// TIA Portal project "SCI_prueba_485" (V17)

(* hardware
DEVICE "ET 200SP station_1"  ET 200SP-Station
   slot 0: "Rack_0"  Rack  6ES5 710-8MAx1
   slot 1: "PLC_1"  CPU 1510SP-1 PN  6ES7 510-1DJ01-0AB0  V2.9
      slot 32768: "Interfaz PROFINET_1"  X1
   slot 2: "CM PtP_1"  CM PtP  6ES7 137-6AA01-0BA0  V2.0
      slot 1: "CM PtP_1"  CM PtP Sub
   slot 3: "Módulo servidor_1"  Server module  6ES7 193-6PA00-0AA0  V1.1
      slot 1: "Módulo servidor_1"  Server module
   slot 127: "BA 2xRJ45"  BA 2xRJ45  6ES7 193-6AR00-0AA0  V0.0
      slot 32769: "Port_1"  6ES7 193-6AR00-0AA0
      slot 32770: "Port_2"  6ES7 193-6AR00-0AA0
*)

// ===== PLC "PLC_1"  CPU 1510SP-1 PN =====

VAR_GLOBAL   // PLC tag table "Tabla de variables estándar"
   "System_Byte" AT %MB1 : Byte;
   "FirstScan" AT %M1.0 : Bool;
   "DiagStatusUpdate" AT %M1.1 : Bool;
   "AlwaysTRUE" AT %M1.2 : Bool;
   "AlwaysFALSE" AT %M1.3 : Bool;
   "Clock_Byte" AT %MB0 : Byte;
   "Clock_10Hz" AT %M0.0 : Bool;
   "Clock_5Hz" AT %M0.1 : Bool;
   "Clock_2.5Hz" AT %M0.2 : Bool;
   "Clock_2Hz" AT %M0.3 : Bool;
   "Clock_1.25Hz" AT %M0.4 : Bool;
   "Clock_1Hz" AT %M0.5 : Bool;
   "Clock_0.625Hz" AT %M0.6 : Bool;
   "Clock_0.5Hz" AT %M0.7 : Bool;
   "Tag_1" AT %MD100 : DWord;
   "Tag_2" AT %M50.0 : Bool;
   "Tag_3" AT %M64.0 : Bool;
   "Tag_4" AT %M64.1 : Bool;
   "Tag_5" AT %M70.0 : Bool;
END_VAR

VAR_GLOBAL   // PLC tag table "IO"
   "ZS01" AT %I0.0 : Bool;   // Contacto Magnético P2-6
   "ZS02" AT %I0.1 : Bool;   // Contacto Magnético P2-5
   "ZS03" AT %I0.2 : Bool;   // Contacto Magnético P2-4
   "HS01" AT %I0.3 : Bool;   // Pulsador P2-6 A
   "HS02" AT %I0.4 : Bool;   // Pulsador P2-6 B
   "HS03" AT %I0.5 : Bool;   // Pulsador P2-5 A
   "HS04" AT %I0.6 : Bool;   // Pulsador P2-4 A
   "HSS01" AT %I0.7 : Bool;   // Puño de emergencia ducha
   "YY01" AT %I1.0 : Bool;   // Señal apertura del controlador puerta P2-5
   "YY02" AT %I1.1 : Bool;   // Señal apertura del controlador puerta P2-4
   "PSH01" AT %I1.2 : Bool;   // Presóstado burlete P2-6
   "E1.3" AT %I1.3 : Bool;   // Reserva
   "E1.4" AT %I1.4 : Bool;   // Reserva
   "E1.5" AT %I1.5 : Bool;   // Reserva
   "E1.6" AT %I1.6 : Bool;   // Reserva
   "E1.7" AT %I1.7 : Bool;   // Reserva
   "EV01" AT %A0.0 : Bool;   // Electroválvula ducha
   "KY01" AT %Q0.1 : Bool;   // PUERTA P2-6
   "KY02" AT %Q0.2 : Bool;   // PUERTA P2-5
   "KY03" AT %Q0.3 : Bool;   // PUERTA P2-4
   "HA01" AT %Q0.4 : Bool;   // P2-6 Buzzer - Hombre atrapado
   "HL01" AT %Q0.5 : Bool;   // P2-6 Lámpara - Falla
   "KY04" AT %Q0.6 : Bool;   // Reinicio fuente
   "Q0.7" AT %Q0.7 : Bool;   // Reserva
   "Q1.0" AT %Q1.0 : Bool;   // Reserva
   "Q1.1" AT %Q1.1 : Bool;   // Reserva
   "Q1.2" AT %Q1.2 : Bool;   // Reserva
   "Q1.3" AT %Q1.3 : Bool;   // Reserva
   "Q1.4" AT %Q1.4 : Bool;   // Reserva
   "Q1.5" AT %Q1.5 : Bool;   // Reserva
   "Q1.6" AT %Q1.6 : Bool;   // Reserva
   "Q1.7" AT %Q1.7 : Bool;   // Reserva
END_VAR

TYPE "FALLAS"
   STRUCT
      PE_FACT : Bool;   // Falla: Emergencia actuada
      Vestuario_FTMO : Bool;   // Falla: Persona en vestuario por demasiado tiempo
      Ducha_FTMO : Bool;   // Falla: Persona en ducha por demasiado tiempo
      "P2-6_FATR" : Bool;   // Falla: P2-6 Persona atrapada
      "P2-5_FATR" : Bool;   // Falla: P2-5 Persona atrapada
      "P2-4_FATR" : Bool;   // Falla: P2-4 Persona atrapada
      "P2-6_TMO_FABR" : Bool;   // Falla: Puerta P2-6 abierta
      "P2-5_TMO_FABR" : Bool;   // Falla: Puerta P2-5 abierta
      "P2-4_TMO_FABR" : Bool;   // Falla: Puerta P2-4 abierta
   END_STRUCT;
END_TYPE

DATA_BLOCK "DB1_AVISOS"   // DB1
TITLE = DB Avisos
{ S7_Optimized_Access := 'FALSE' }
AUTHOR : IGLP
VERSION : 0.1
   VAR
      PRE : "FALLAS";
      MEM : "FALLAS";
      REC : "FALLAS";
      CMD : "FALLAS";
      CMD_AUX : "FALLAS";
      CMD_FLA : "FALLAS";
   END_VAR
BEGIN
END_DATA_BLOCK

DATA_BLOCK "DB2_CODIGOS"   // DB2
TITLE = Códigos habilitados
{ S7_Optimized_Access := 'TRUE' }
AUTHOR : IGLP
VERSION : 0.1
   VAR
      PIN_Nuevo_TCL1 : Bool;
      PIN_Nuevo_TCL2 : Bool;
      PIN_TCL1_OK : Bool;
      PIN_TCL2_OK : Bool;
      PIN_TCL1_ERR : Bool;
      PIN_TCL2_ERR : Bool;
      PIN_Codigo_TCL1 : Int;
      PIN_Codigo_TCL2 : Int;
      PIN_Codigo_TCL1_OK : Int;
      PIN_Codigo_TCL2_OK : Int;
      Aux_inidice : Int;
      TCL1_TMR_BitVida : IEC_TIMER;
      TCL2_TMR_BitVida : IEC_TIMER;
      TCL_TMR_ESP : IEC_TIMER;
      TCL_PWR_OFF : IEC_TIMER;
   END_VAR
   VAR RETAIN
      PIN : Array[0..500] of Int;
   END_VAR
BEGIN
END_DATA_BLOCK

DATA_BLOCK "DB3_GRAL"   // DB3
TITLE = DB Comandos eléctricos
{ S7_Optimized_Access := 'TRUE' }
VERSION : 0.1
   VAR
      MODO : Int;   // Modo: 0 - Manual / 1 Automático
      REINICIO : Int;
      SILENCIAR : Int;
      CNT_Personas : Int;
      CNT_HS01 : Int;   // P2-6A: Cantidad de veces pulsado
      CNT_HS02 : Int;   // P2-6B: Cantidad de veces pulsado
      CNT_HS03 : Int;   // P2-5A: Cantidad de veces pulsado
      CNT_HS04 : Int;   // P2-4A: Cantidad de veces pulsado
      SFA : Bool;   // Sin fallas
      FNUE : Bool;   // Falla nueva
      FPRE : Bool;   // Falla presente
      "P2-x_ResFal" : Bool;   // Resumen de fallas de puerta
      fpHS01 : Bool;   // Flanco positivo - Pulsador P2-6 A
      fpHS02 : Bool;   // Flanco positivo - Pulsador P2-6 B
      fpHS03 : Bool;   // Flanco positivo - Pulsador P2-5 A
      fpHS04 : Bool;   // Flanco positivo - Pulsador P2-4 A
      xHS01 : Bool;
      xHS02 : Bool;
      xHS03 : Bool;
      xHS04 : Bool;
      xZS01 : Bool;
      xZS02 : Bool;
      xZS03 : Bool;
      xS161 : Bool;
      xS261 : Bool;
      TMR_TMO_Vestuario : IEC_TIMER;
      TMR_TMO_Ducha : IEC_TIMER;
      "TMR_P2-6_CRR" : IEC_TIMER;
      "TMR_P2-5_CRR" : IEC_TIMER;
      "TMR_P2-4_CRR" : IEC_TIMER;
      TMR_HS01_SCADA : IEC_TIMER;
      TMR_HS02_SCADA : IEC_TIMER;
      TMR_HS03_SCADA : IEC_TIMER;
      TMR_HS04_SCADA : IEC_TIMER;
      TMR_ZS01 : IEC_TIMER;
      TMR_ZS02 : IEC_TIMER;
      TMR_ZS03 : IEC_TIMER;
      TMR_PSH01 : IEC_TIMER;
      ZS01_TMP : Bool;   // Contacto Magnético P2-6 - Temporizado
      ZS02_TMP : Bool;   // Contacto Magnético P2-5 - Temporizado
      ZS03_TMP : Bool;   // Contacto Magnético P2-4 - Temporizado
      PSH01_TMP : Bool;   // Presóstado burlete P2-6 - Temporizado
      "P2-6" : Struct   // Puerta Pasillo <-> Vestuario P2-6
         TMR_Sol_Man : IEC_TIMER;
         Sol_Man : Bool;   // Solicitud manual de apertura
         HW : Bool;   // Hardware Interlock
         CMD : Bool;   // Comando de apertura
      END_STRUCT;
      "P2-5" : Struct   // Puerta Vestuario <-> Ducha P2-5
         TMR_Sol_Man : IEC_TIMER;
         Sol_Man : Bool;   // Solicitud manual de apertura
         HW : Bool;   // Hardware Interlock
         CMD : Bool;   // Comando de apertura
      END_STRUCT;
      "P2-4" : Struct   // Puerta Ducha <-> Bioterio P2-4
         TMR_Sol_Man : IEC_TIMER;
         Sol_Man : Bool;   // Solicitud manual de apertura
         HW : Bool;   // Hardware Interlock
         CMD : Bool;   // Comando de apertura
      END_STRUCT;
      Ducha : Struct   // Ducha - Electroválvula
         TMR_Sol_Man : IEC_TIMER;
         Sol_Man : Bool;   // Solicitud manual de apertura
         HW : Bool;   // Hardware Interlock
         CMD : Bool;
      END_STRUCT;
   END_VAR
BEGIN
END_DATA_BLOCK

DATA_BLOCK "DB10_Parámetros"   // DB10
TITLE = DB Parametros del sistema
{ S7_Optimized_Access := 'TRUE' }
AUTHOR : IGLP
VERSION : 0.1
   VAR RETAIN
      SP_N_APA : Int := 10;   // Consigna de veces antes de aviso persona atrapada
      SP_Tmp_Ducha_1 : DInt;   // Consigna de tiempo de ducha activa [ms]
      SP_Tmp_Ducha_2 : DInt := 30000;   // Consigna de tiempo de ducha activa [ms]
      SP_Tmp_Ducha_Pre : DInt;   // Consigna de tiempo de precalentar ducha [ms]
      SP_TMO_Ducha : DInt;   // Consigna de tiempo en ducha [ms]
      SP_TMO_Vestuario : DInt;   // Consigna de tiempo en vestuario [ms]
      SP_TMO_PTA_ABR : DInt;   // Consigna de tiempo alarma puerta abierta [ms]
   END_VAR
BEGIN
END_DATA_BLOCK

DATA_BLOCK "DB20_Modbus_Config"   // DB20
{ S7_Optimized_Access := 'TRUE' }
VERSION : 0.1
   VAR
      TC_NDR : Bool := FALSE;
      TC_DR : Bool := FALSE;
      TC_Error : Bool := FALSE;
      TC_Status : Word := 16#7000;
      SCADA_NDR : Bool := FALSE;
      SCADA_DR : Bool := FALSE;
      SCADA_Error : Bool := TRUE;
      SCADA_Status : Word := 16#8389;
      DATA : Array[0..1] of Int;
      SCADA_CONN : TCON_IP_v4;
   END_VAR
BEGIN
   SCADA_CONN.InterfaceId := 64;
   SCADA_CONN.ID := 16#001E;
   SCADA_CONN.ConnectionType := 16#0B;
   SCADA_CONN.LocalPort := 502;
   SCADA_CONN.RemotePort := 0;
   SCADA_CONN.ActiveEstablished := FALSE;
   SCADA_CONN.RemoteAddress.ADDR[1] := 0;
   SCADA_CONN.RemoteAddress.ADDR[2] := 0;
   SCADA_CONN.RemoteAddress.ADDR[3] := 0;
   SCADA_CONN.RemoteAddress.ADDR[4] := 0;
END_DATA_BLOCK

DATA_BLOCK "DB21_Modbus_Data_1"   // DB21
{ S7_Optimized_Access := 'FALSE' }
VERSION : 0.1
   VAR
      "NBS 3A" : Struct
         Modo : Int;   // Scada -> PLC: Modo (0-Manual / 1-Automático)
         Reinicio : Int;   // Scada -> PLC: Reset de secuencia
         Silenciar : Int;   // Scada -> PLC: Silenciar alarma
         SP_Tmp_Ducha : Int;   // Scada -> PLC: Consigna de tiempo de ducha activa [s]
         SP_Tmp_Ducha_Pre : Int;   // Scada -> PLC: Consigna de tiempo de precalentar ducha [s]
         SP_TMO_Ducha : Int;   // Scada -> PLC: Consigna de tiempo en ducha [s]
         SP_TMO_Vestuario : Int;   // Scada -> PLC: Consigna de tiempo en vestuario [s]
         SP_TMO_PTA_ABR : Int;   // Scada -> PLC: Consigna de tiempo alarma puerta abierta [s]
         CNT_Personas : Int;   // PLC -> Scada: Contador de personas dentro de bioterio
         "P2-6_Est" : Int;   // PLC -> Scada: P2-6 - Puerta Pasillo: Estado (0-Cerrada / 1-Abierta / 2-Falla reconocida / 3-Falla nueva)
         "P2-5_Est" : Int;   // PLC -> Scada: P2-5 - Puerta Ducha Ingreso: Estado (0-Cerrada / 1-Abierta / 2-Falla reconocida / 3-Falla nueva)
         "P2-4_Est" : Int;   // PLC -> Scada: P2-4 - Puerta Ducha Salida: Estado (0-Cerrada / 1-Abierta / 2-Falla reconocida / 3-Falla nueva)
         HSS01_Est : Int;   // PLC -> Scada: Pulsador de Emergencia en Ducha (0-Normal/ 1-Activada/ 2-Falla reconocida / 3-Falla nueva)
         HS01_Est : Int;   // PLC -> Scada: P2-6A: Pulsador Ingreso (0-Normal / 1-Presionado)
         HS02_Est : Int;   // PLC -> Scada: P2-6B: Pulsador Salida (0-Normal / 1-Presionado)
         HS03_Est : Int;   // PLC -> Scada: P2-5A: Pulsador Ducha Ingreso (0-Normal / 1-Presionado)
         HS04_Est : Int;   // PLC -> Scada: P2-4A: Pulsador Ducha Salida (0-Normal / 1-Presionado)
         EV01_Est : Int;   // PLC -> Scada: Ducha: Electroválvula (0-Normal/ 1-Activada/ 2-Falla reconocida / 3-Falla nueva)
         TCL01_PIN : Int;   // PLC -> Scada: P2-5: PIN ingresado en teclado
         TCL02_PIN : Int;   // PLC -> Scada: P2-6: PIN ingresado en teclado
         Ducha_PIN : Int;   // PLC -> Scada: Ducha: PIN de quien ingresó a ducha
         Vesuario_Est : Int;   // PLC -> Scada: Vestuario: Estado (0-Desocupado / 1-Ocupado / 2-Falla reconocida / 3-Falla nueva)
         Ducha_Est : Int;   // PLC -> Scada: Ducha: Estado (0-Desocupada / 1-Ocupada / 2-Falla reconocida / 3-Falla nueva)
         Alarma : Int;   // PLC -> Scada: Resumen de alarmas (0-Sin alarma / 1-Alarma presente)
      END_STRUCT;
   END_VAR
BEGIN
END_DATA_BLOCK

DATA_BLOCK "DB22_Modbus_Data_2"   // DB22
{ S7_Optimized_Access := 'FALSE' }
VERSION : 0.1
   VAR
      CODIGOS : Array[1..100] of Int;
   END_VAR
BEGIN
END_DATA_BLOCK

DATA_BLOCK "DB23_Modbus_Data_3"   // DB23
{ S7_Optimized_Access := 'FALSE' }
VERSION : 0.1
   VAR
      data : Array[0..10] of Int;
      TCL : Struct
         "TCL1 P2-5 PIN" : Int;
         "TCL1 P2-5 ALIVE" : Int;
         "TCL2 P2-4 PIN" : Int;
         "TCL2 P2-4 ALIVE" : Int;
      END_STRUCT;
   END_VAR
BEGIN
END_DATA_BLOCK

DATA_BLOCK "DB50_Secuencia"   // DB50
{ S7_Optimized_Access := 'TRUE' }
VERSION : 0.1
// stored: InstanceOfName Secuencia
"Secuencia"
BEGIN
END_DATA_BLOCK

DATA_BLOCK "DB51_Transiciones"   // DB51
TITLE = DB Transiciones y estados del secuencial
{ S7_Optimized_Access := 'TRUE' }
AUTHOR : IGLP
VERSION : 0.1
   VAR
      TMR_Puerta : IEC_TIMER;
      TMR_DUCHA_ESP_INI : IEC_TIMER;
      TMR_DUCHA_PRE : IEC_TIMER;
      TMR_DUCHA_1 : IEC_TIMER;
      TMR_DUCHA_2 : IEC_TIMER;
      TMR_DUCHA_3 : IEC_TIMER;
   END_VAR
   VAR RETAIN
      S : Struct
         "10" : Bool;   // Reposo
         "110" : Bool;   // Ingreso a bioterio: Solicitud ingreso Pasillo -> Vestuario
         "111" : Bool;   // Ingreso a bioterio: Puerta P2-6 abierta
         "120" : Bool;   // Ingreso a bioterio: Vestuario ocupado
         "121" : Bool;   // Ingreso a bioterio: Solicitud de precalentar ducha
         "130" : Bool;   // Ingreso a bioterio: Solicitud salir Vestuario -> Pasillo
         "131" : Bool;   // Ingreso a bioterio: Puerta P2-6 abierta
         "140" : Bool;   // Ingreso a bioterio: Solicitud ingreso Vestuario -> Ducha
         "141" : Bool;   // Ingreso a bioterio: Puerta P2-5 abierta
         "150" : Bool;   // Ingreso a bioterio: Ducha ocupada
         "160" : Bool;   // Ingreso a bioterio: Solicitud salir Ducha -> Bioterio
         "161" : Bool;   // Ingreso a bioterio: Puerta P2-4 abierta
         "170" : Bool;   // Ingreso a bioterio: Solicitud salir Ducha -> Vestuario
         "171" : Bool;   // Ingreso a bioterio: Puerta P2-5 abierta
         "210" : Bool;   // Egreso de bioterio: Solicitud ingreso Bioterio -> Ducha
         "211" : Bool;   // Egreso de bioterio: Puerta P2-4 abierta
         "220" : Bool;   // Egreso de bioterio: Ducha ocupada - Espera incial
         "221" : Bool;   // Egreso de bioterio: Ducha ocupada - Válvula abierta
         "222" : Bool;   // Egreso de bioterio: Ducha ocupada - Pausa ducha
         "223" : Bool;   // Egreso de bioterio: Ducha ocupada - Válvula abierta
         "224" : Bool;   // Egreso de bioterio: Ducha ocupada
         "230" : Bool;   // Egreso de bioterio: Solicitud salir Ducha -> Bioterio
         "231" : Bool;   // Egreso de bioterio: Puerta P2-4 abierta
         "240" : Bool;   // Egreso de bioterio: Solicitud salir Ducha -> Vestuario
         "241" : Bool;   // Egreso de bioterio: Puerta P2-5 abierta
         "250" : Bool;   // Egreso de bioterio: Vestuario ocupado
         "251" : Bool;   // Egreso de bioterio: Solicitud de precalentar ducha
         "260" : Bool;   // Egreso de bioterio: Solicitud salir Vestuario -> Pasillo
         "261" : Bool;   // Egreso de bioterio: Puerta P2-6 abierta
         "270" : Bool;   // Egreso de bioterio: Solicitud ingreso Vestuario -> Ducha
         "271" : Bool;   // Egreso de bioterio: Puerta P2-5 abierta
         "310" : Bool;   // Egreso de bioterio: Solicitud de precalentar ducha
      END_STRUCT;
   END_VAR
   VAR
      T : Struct
         T10_110 : Bool;
         T110_111 : Bool;
         T111_120 : Bool;
         T110_10 : Bool;
         T120_121 : Bool;
         T121_120 : Bool;
         T120_140 : Bool;
         T140_141 : Bool;
         T120_130 : Bool;
         T130_131 : Bool;
         T130_120 : Bool;
         T131_10 : Bool;
         T141_150 : Bool;
         T150_160 : Bool;
         T160_161 : Bool;
         T160_150 : Bool;
         T161_10 : Bool;
         T150_170 : Bool;
         T170_171 : Bool;
         T171_120 : Bool;
         T170_150 : Bool;
         T10_210 : Bool;
         T210_211 : Bool;
         T211_220 : Bool;
         T220_221 : Bool;
         T221_222 : Bool;
         T222_223 : Bool;
         T223_224 : Bool;
         T224_230 : Bool;
         T224_240 : Bool;
         T240_241 : Bool;
         T241_250 : Bool;
         T240_224 : Bool;
         T250_260 : Bool;
         T260_261 : Bool;
         T261_10 : Bool;
         T260_250 : Bool;
         T250_270 : Bool;
         T270_271 : Bool;
         T271_224 : Bool;
         T270_250 : Bool;
         T250_251 : Bool;
         T251_250 : Bool;
         T210_10 : Bool;
         T220_230 : Bool;
         T230_231 : Bool;
         T230_220 : Bool;
         T231_10 : Bool;
         T10_310 : Bool;
         T310_10 : Bool;
      END_STRUCT;
   END_VAR
BEGIN
END_DATA_BLOCK

FUNCTION_BLOCK "Secuencia"   // FB1, GRAPH_PLUS
{ S7_Optimized_Access := 'TRUE' }
VERSION : 0.1
   VAR_INPUT
      OFF_SQ : Bool := false;   // Desactivar cadena
      INIT_SQ : Bool := false;   // Poner cadena en estado inicial
      ACK_EF : Bool := false;   // Acusar todos los errores y fallos
      S_PREV : Bool := false;   // Mostrar la etapa anterior en el parámetro S_NO
      S_NEXT : Bool := false;   // Mostrar la etapa siguiente en el parámetro S_NO
      SW_AUTO : Bool := false;   // Modo automático
      SW_TAP : Bool := false;   // Semiautomático/continuar con transición
      SW_TOP : Bool := false;   // Semiautomático/transición ignorada
      SW_MAN : Bool := false;   // Modo manual
      S_SEL : Int := 0;   // Seleccionar la etapa que debe mostrarse en S_NO
      S_ON : Bool := false;   // Activar la etapa del parámetro S_NO
      S_OFF : Bool := false;   // Desactivar el incremento presente en el parámetro S_NO
      T_PUSH : Bool := false;   // Habilitar conmutación de transición en modo semiautomático
   END_VAR
   VAR_OUTPUT
      S_NO : Int := 0;   // Número de etapa
      S_MORE : Bool := false;   // Existen más etapas que pueden mostrarse en S_NO.
      S_ACTIVE : Bool := false;   // El incremento presente en el parámetro S_NO está activo
      ERR_FLT : Bool := false;   // Error de grupo interlock o supervisión
      AUTO_ON : Bool := false;   // Modo automático activado
      TAP_ON : Bool := false;   // Modo semiautomático/etapa con transición activada
      TOP_ON : Bool := false;   // Modo semiautomático/Ignorar transición activado
      MAN_ON : Bool := false;   // Modo manual activado
   END_VAR
   VAR
      HMI_INFO : Array[0..8] of UInt;
      IF_PAR : G7_IfParPlus_V6;
      RT_DATA : G7_RTDataPlus_V6;   // Área de datos interna
      T10_110 : G7_TransitionPlus_V6;   // Estructura de la transición
      T110_111 : G7_TransitionPlus_V6;   // Estructura de la transición
      T111_120 : G7_TransitionPlus_V6;   // Estructura de la transición
      T120_140 : G7_TransitionPlus_V6;   // Estructura de la transición
      T140_141 : G7_TransitionPlus_V6;   // Estructura de la transición
      T141_150 : G7_TransitionPlus_V6;   // Estructura de la transición
      T150_160 : G7_TransitionPlus_V6;   // Estructura de la transición
      T160_161 : G7_TransitionPlus_V6;   // Estructura de la transición
      T120_121 : G7_TransitionPlus_V6;   // Estructura de la transición
      T121_120 : G7_TransitionPlus_V6;   // Estructura de la transición
      T120_130 : G7_TransitionPlus_V6;   // Estructura de la transición
      T130_131 : G7_TransitionPlus_V6;   // Estructura de la transición
      T161_10 : G7_TransitionPlus_V6;   // Estructura de la transición
      T160_150 : G7_TransitionPlus_V6;   // Estructura de la transición
      T150_170 : G7_TransitionPlus_V6;   // Estructura de la transición
      T170_171 : G7_TransitionPlus_V6;   // Estructura de la transición
      T170_120 : G7_TransitionPlus_V6;   // Estructura de la transición
      T170_150 : G7_TransitionPlus_V6;   // Estructura de la transición
      T130_120 : G7_TransitionPlus_V6;   // Estructura de la transición
      T131_10 : G7_TransitionPlus_V6;   // Estructura de la transición
      T10_210 : G7_TransitionPlus_V6;   // Estructura de la transición
      T210_211 : G7_TransitionPlus_V6;   // Estructura de la transición
      T211_220 : G7_TransitionPlus_V6;   // Estructura de la transición
      T220_221 : G7_TransitionPlus_V6;   // Estructura de la transición
      T221_222 : G7_TransitionPlus_V6;   // Estructura de la transición
      T222_223 : G7_TransitionPlus_V6;   // Estructura de la transición
      T223_224 : G7_TransitionPlus_V6;   // Estructura de la transición
      T224_240 : G7_TransitionPlus_V6;   // Estructura de la transición
      S220_230 : G7_TransitionPlus_V6;   // Estructura de la transición
      S230_231 : G7_TransitionPlus_V6;   // Estructura de la transición
      T231_10 : G7_TransitionPlus_V6;   // Estructura de la transición
      S230_220 : G7_TransitionPlus_V6;   // Estructura de la transición
      T210_10 : G7_TransitionPlus_V6;   // Estructura de la transición
      T240_241 : G7_TransitionPlus_V6;   // Estructura de la transición
      T260_261 : G7_TransitionPlus_V6;   // Estructura de la transición
      T241_250 : G7_TransitionPlus_V6;   // Estructura de la transición
      T250_260 : G7_TransitionPlus_V6;   // Estructura de la transición
      T261_10 : G7_TransitionPlus_V6;   // Estructura de la transición
      T250_270 : G7_TransitionPlus_V6;   // Estructura de la transición
      T270_271 : G7_TransitionPlus_V6;   // Estructura de la transición
      T271_224 : G7_TransitionPlus_V6;   // Estructura de la transición
      T270_250 : G7_TransitionPlus_V6;   // Estructura de la transición
      T250_251 : G7_TransitionPlus_V6;   // Estructura de la transición
      T251_250 : G7_TransitionPlus_V6;   // Estructura de la transición
      T10_310 : G7_TransitionPlus_V6;   // Estructura de la transición
      T310_10 : G7_TransitionPlus_V6;   // Estructura de la transición
      T110_10 : G7_TransitionPlus_V6;   // Estructura de la transición
      T240_224 : G7_TransitionPlus_V6;   // Estructura de la transición
      T260_250 : G7_TransitionPlus_V6;   // Estructura de la transición
      T224_230 : G7_TransitionPlus_V6;   // Estructura de la transición
      Reposo : G7_StepPlus_V6;   // Estructura de la etapa
      S110 : G7_StepPlus_V6;   // Estructura de la etapa
      S111 : G7_StepPlus_V6;   // Estructura de la etapa
      S120 : G7_StepPlus_V6;   // Estructura de la etapa
      S121 : G7_StepPlus_V6;   // Estructura de la etapa
      S130 : G7_StepPlus_V6;   // Estructura de la etapa
      S131 : G7_StepPlus_V6;   // Estructura de la etapa
      S140 : G7_StepPlus_V6;   // Estructura de la etapa
      S141 : G7_StepPlus_V6;   // Estructura de la etapa
      S150 : G7_StepPlus_V6;   // Estructura de la etapa
      S160 : G7_StepPlus_V6;   // Estructura de la etapa
      S161 : G7_StepPlus_V6;   // Estructura de la etapa
      S170 : G7_StepPlus_V6;   // Estructura de la etapa
      S171 : G7_StepPlus_V6;   // Estructura de la etapa
      S210 : G7_StepPlus_V6;   // Estructura de la etapa
      S211 : G7_StepPlus_V6;   // Estructura de la etapa
      S220 : G7_StepPlus_V6;   // Estructura de la etapa
      S221 : G7_StepPlus_V6;   // Estructura de la etapa
      S222 : G7_StepPlus_V6;   // Estructura de la etapa
      S223 : G7_StepPlus_V6;   // Estructura de la etapa
      S224 : G7_StepPlus_V6;   // Estructura de la etapa
      S230 : G7_StepPlus_V6;   // Estructura de la etapa
      S231 : G7_StepPlus_V6;   // Estructura de la etapa
      S240 : G7_StepPlus_V6;   // Estructura de la etapa
      S241 : G7_StepPlus_V6;   // Estructura de la etapa
      S250 : G7_StepPlus_V6;   // Estructura de la etapa
      S251 : G7_StepPlus_V6;   // Estructura de la etapa
      S260 : G7_StepPlus_V6;   // Estructura de la etapa
      S261 : G7_StepPlus_V6;   // Estructura de la etapa
      S270 : G7_StepPlus_V6;   // Estructura de la etapa
      S271 : G7_StepPlus_V6;   // Estructura de la etapa
      S310 : G7_StepPlus_V6;   // Estructura de la etapa
      SINI : Array[0..1] of USInt;
      LSTT : Array[0..49] of USInt;
      ATAJ : Array[0..49] of USInt;
      ATAB : Array[0..49] of USInt;
      PSTT : Array[0..49] of USInt;
      NSTT : Array[0..49] of USInt;
      ASSJ : Array[0..31] of USInt;
      ASSB : Array[0..31] of USInt;
      PTTS : Array[0..31] of USInt;
      NTTS : Array[0..31] of USInt;
      SW_SQTS : Array[0..31] of USInt;
      SWITCH : Array[0..71] of USInt;
      TVX : Array[0..34] of USInt;
      TTX : Array[0..34] of USInt;
      TSX : Array[0..1] of USInt;
      S00X : Array[0..1] of USInt;
      SOFFX : Array[0..1] of USInt;
      SONX : Array[0..1] of USInt;
      SAX : Array[0..1] of USInt;
      SERRX : Array[0..32] of USInt;
      SMX : Array[0..32] of USInt;
      S0X : Array[0..32] of USInt;
      S1X : Array[0..32] of USInt;
      IL_ALARM_INST : Diag_Alarm;
      SUP_ALARM_INST : Diag_Alarm;
      STEP_TIME_ALARM_INST : Diag_Alarm;
      IEC_TIMER_INST : IEC_TIMER;
      TRANSACTION_FLAG : Bool := false;
   END_VAR
   // SINI[0] := 2;
   // LSTT[0] := 255;
   // LSTT[1] := 255;
   // LSTT[2] := 255;
   // LSTT[3] := 255;
   // LSTT[4] := 255;
   // LSTT[5] := 255;
   // LSTT[6] := 255;
   // LSTT[7] := 255;
   // LSTT[8] := 255;
   // LSTT[9] := 3;
   // LSTT[10] := 255;
   // LSTT[11] := 255;
   // LSTT[13] := 9;
   // LSTT[14] := 255;
   // LSTT[15] := 255;
   // LSTT[16] := 3;
   // LSTT[17] := 9;
   // LSTT[18] := 3;
   // LSTT[20] := 255;
   // LSTT[21] := 255;
   // LSTT[22] := 255;
   // LSTT[23] := 255;
   // LSTT[24] := 255;
   // LSTT[25] := 255;
   // LSTT[26] := 255;
   // LSTT[27] := 255;
   // LSTT[28] := 255;
   // LSTT[29] := 255;
   // LSTT[31] := 16;
   // LSTT[33] := 255;
   // LSTT[34] := 255;
   // LSTT[35] := 255;
   // LSTT[36] := 255;
   // LSTT[38] := 255;
   // LSTT[39] := 255;
   // LSTT[40] := 20;
   // LSTT[41] := 25;
   // LSTT[42] := 255;
   // LSTT[43] := 25;
   // LSTT[44] := 255;
   // ATAJ[1] := 1;
   // ATAJ[2] := 2;
   // ATAJ[3] := 3;
   // ATAJ[4] := 4;
   // ATAJ[5] := 5;
   // ATAJ[6] := 6;
   // ATAJ[7] := 7;
   // ATAJ[8] := 8;
   // ATAJ[9] := 9;
   // ATAJ[10] := 10;
   // ATAJ[11] := 11;
   // ATAJ[12] := 12;
   // ATAJ[13] := 13;
   // ATAJ[14] := 14;
   // ATAJ[15] := 15;
   // ATAJ[16] := 16;
   // ATAJ[17] := 17;
   // ATAJ[18] := 18;
   // ATAJ[19] := 19;
   // ATAJ[20] := 20;
   // ATAJ[21] := 21;
   // ATAJ[22] := 22;
   // ATAJ[23] := 23;
   // ATAJ[24] := 24;
   // ATAJ[25] := 25;
   // ATAJ[26] := 26;
   // ATAJ[27] := 27;
   // ATAJ[28] := 28;
   // ATAJ[29] := 29;
   // ATAJ[30] := 30;
   // ATAJ[31] := 31;
   // ATAJ[32] := 32;
   // ATAJ[33] := 33;
   // ATAJ[34] := 34;
   // ATAJ[35] := 35;
   // ATAJ[36] := 36;
   // ATAJ[37] := 37;
   // ATAJ[38] := 38;
   // ATAJ[39] := 39;
   // ATAJ[40] := 40;
   // ATAJ[41] := 41;
   // ATAJ[42] := 42;
   // ATAJ[43] := 43;
   // ATAJ[44] := 44;
   // ATAJ[45] := 45;
   // ATAB[0] := 20;
   // ATAB[1] := 46;
   // ATAB[2] := 2;
   // ATAB[3] := 8;
   // ATAB[4] := 4;
   // ATAB[5] := 5;
   // ATAB[6] := 14;
   // ATAB[7] := 13;
   // ATAB[8] := 10;
   // ATAB[9] := 9;
   // ATAB[10] := 3;
   // ATAB[11] := 18;
   // ATAB[12] := 12;
   // ATAB[13] := 7;
   // ATAB[14] := 6;
   // ATAB[15] := 17;
   // ATAB[16] := 16;
   // ATAB[17] := 15;
   // ATAB[18] := 11;
   // ATAB[19] := 19;
   // ATAB[20] := 44;
   // ATAB[21] := 32;
   // ATAB[22] := 22;
   // ATAB[23] := 28;
   // ATAB[24] := 24;
   // ATAB[25] := 25;
   // ATAB[26] := 26;
   // ATAB[27] := 49;
   // ATAB[28] := 23;
   // ATAB[29] := 31;
   // ATAB[30] := 30;
   // ATAB[31] := 29;
   // ATAB[32] := 21;
   // ATAB[33] := 47;
   // ATAB[34] := 48;
   // ATAB[35] := 35;
   // ATAB[36] := 38;
   // ATAB[37] := 37;
   // ATAB[38] := 42;
   // ATAB[39] := 41;
   // ATAB[40] := 40;
   // ATAB[41] := 39;
   // ATAB[42] := 36;
   // ATAB[43] := 43;
   // ATAB[45] := 45;
   // PSTT[1] := 1;
   // PSTT[2] := 2;
   // PSTT[3] := 3;
   // PSTT[4] := 7;
   // PSTT[5] := 8;
   // PSTT[6] := 9;
   // PSTT[7] := 10;
   // PSTT[8] := 3;
   // PSTT[9] := 4;
   // PSTT[10] := 3;
   // PSTT[11] := 5;
   // PSTT[12] := 11;
   // PSTT[13] := 10;
   // PSTT[14] := 9;
   // PSTT[15] := 12;
   // PSTT[16] := 13;
   // PSTT[17] := 12;
   // PSTT[18] := 5;
   // PSTT[19] := 6;
   // PSTT[21] := 14;
   // PSTT[22] := 15;
   // PSTT[23] := 16;
   // PSTT[24] := 17;
   // PSTT[25] := 18;
   // PSTT[26] := 19;
   // PSTT[27] := 20;
   // PSTT[28] := 16;
   // PSTT[29] := 21;
   // PSTT[30] := 22;
   // PSTT[31] := 21;
   // PSTT[32] := 14;
   // PSTT[33] := 23;
   // PSTT[34] := 27;
   // PSTT[35] := 24;
   // PSTT[36] := 25;
   // PSTT[37] := 28;
   // PSTT[38] := 25;
   // PSTT[39] := 29;
   // PSTT[40] := 30;
   // PSTT[41] := 29;
   // PSTT[42] := 25;
   // PSTT[43] := 26;
   // PSTT[45] := 31;
   // NSTT[0] := 1;
   // NSTT[1] := 2;
   // NSTT[2] := 3;
   // NSTT[3] := 7;
   // NSTT[4] := 8;
   // NSTT[5] := 9;
   // NSTT[6] := 10;
   // NSTT[7] := 11;
   // NSTT[8] := 4;
   // NSTT[9] := 3;
   // NSTT[10] := 5;
   // NSTT[11] := 6;
   // NSTT[13] := 9;
   // NSTT[14] := 12;
   // NSTT[15] := 13;
   // NSTT[16] := 3;
   // NSTT[17] := 9;
   // NSTT[18] := 3;
   // NSTT[20] := 14;
   // NSTT[21] := 15;
   // NSTT[22] := 16;
   // NSTT[23] := 17;
   // NSTT[24] := 18;
   // NSTT[25] := 19;
   // NSTT[26] := 20;
   // NSTT[27] := 23;
   // NSTT[28] := 21;
   // NSTT[29] := 22;
   // NSTT[31] := 16;
   // NSTT[33] := 24;
   // NSTT[34] := 28;
   // NSTT[35] := 25;
   // NSTT[36] := 27;
   // NSTT[38] := 29;
   // NSTT[39] := 30;
   // NSTT[40] := 20;
   // NSTT[41] := 25;
   // NSTT[42] := 26;
   // NSTT[43] := 25;
   // NSTT[44] := 31;
   // ASSJ[1] := 1;
   // ASSJ[2] := 2;
   // ASSJ[3] := 3;
   // ASSJ[4] := 4;
   // ASSJ[5] := 5;
   // ASSJ[6] := 6;
   // ASSJ[7] := 7;
   // ASSJ[8] := 8;
   // ASSJ[9] := 9;
   // ASSJ[10] := 10;
   // ASSJ[11] := 11;
   // ASSJ[12] := 12;
   // ASSJ[13] := 13;
   // ASSJ[14] := 14;
   // ASSJ[15] := 15;
   // ASSJ[16] := 16;
   // ASSJ[17] := 17;
   // ASSJ[18] := 18;
   // ASSJ[19] := 19;
   // ASSJ[20] := 20;
   // ASSJ[21] := 21;
   // ASSJ[22] := 22;
   // ASSJ[23] := 23;
   // ASSJ[24] := 24;
   // ASSJ[25] := 25;
   // ASSJ[26] := 26;
   // ASSJ[27] := 27;
   // ASSJ[28] := 28;
   // ASSJ[29] := 29;
   // ASSJ[30] := 30;
   // ASSJ[31] := 31;
   // ASSB[1] := 1;
   // ASSB[2] := 2;
   // ASSB[3] := 3;
   // ASSB[4] := 4;
   // ASSB[5] := 5;
   // ASSB[6] := 6;
   // ASSB[7] := 7;
   // ASSB[8] := 8;
   // ASSB[9] := 9;
   // ASSB[10] := 10;
   // ASSB[11] := 11;
   // ASSB[12] := 12;
   // ASSB[13] := 13;
   // ASSB[14] := 14;
   // ASSB[15] := 15;
   // ASSB[16] := 16;
   // ASSB[17] := 17;
   // ASSB[18] := 18;
   // ASSB[19] := 19;
   // ASSB[20] := 20;
   // ASSB[21] := 21;
   // ASSB[22] := 22;
   // ASSB[23] := 23;
   // ASSB[24] := 24;
   // ASSB[25] := 25;
   // ASSB[26] := 26;
   // ASSB[27] := 27;
   // ASSB[28] := 28;
   // ASSB[29] := 29;
   // ASSB[30] := 30;
   // ASSB[31] := 31;
   // PTTS[0] := 255;
   // PTTS[2] := 1;
   // PTTS[3] := 2;
   // PTTS[4] := 8;
   // PTTS[5] := 10;
   // PTTS[6] := 11;
   // PTTS[7] := 3;
   // PTTS[8] := 4;
   // PTTS[9] := 5;
   // PTTS[10] := 6;
   // PTTS[11] := 7;
   // PTTS[12] := 14;
   // PTTS[13] := 15;
   // PTTS[14] := 20;
   // PTTS[15] := 21;
   // PTTS[16] := 22;
   // PTTS[17] := 23;
   // PTTS[18] := 24;
   // PTTS[19] := 25;
   // PTTS[20] := 26;
   // PTTS[21] := 28;
   // PTTS[22] := 29;
   // PTTS[23] := 27;
   // PTTS[24] := 33;
   // PTTS[25] := 35;
   // PTTS[26] := 42;
   // PTTS[27] := 36;
   // PTTS[28] := 34;
   // PTTS[29] := 38;
   // PTTS[30] := 39;
   // PTTS[31] := 44;
   // NTTS[1] := 1;
   // NTTS[2] := 2;
   // NTTS[3] := 3;
   // NTTS[4] := 9;
   // NTTS[5] := 11;
   // NTTS[6] := 19;
   // NTTS[7] := 4;
   // NTTS[8] := 5;
   // NTTS[9] := 6;
   // NTTS[10] := 7;
   // NTTS[11] := 12;
   // NTTS[12] := 15;
   // NTTS[13] := 16;
   // NTTS[14] := 21;
   // NTTS[15] := 22;
   // NTTS[16] := 23;
   // NTTS[17] := 24;
   // NTTS[18] := 25;
   // NTTS[19] := 26;
   // NTTS[20] := 27;
   // NTTS[21] := 29;
   // NTTS[22] := 30;
   // NTTS[23] := 33;
   // NTTS[24] := 35;
   // NTTS[25] := 36;
   // NTTS[26] := 43;
   // NTTS[27] := 34;
   // NTTS[28] := 37;
   // NTTS[29] := 39;
   // NTTS[30] := 40;
   // NTTS[31] := 45;
   // SW_SQTS[1] := 1;
   // SW_SQTS[2] := 2;
   // SW_SQTS[3] := 2;
   // SW_SQTS[4] := 3;
   // SW_SQTS[5] := 4;
   // SW_SQTS[6] := 5;
   // SW_SQTS[7] := 6;
   // SW_SQTS[8] := 6;
   // SW_SQTS[9] := 6;
   // SW_SQTS[10] := 7;
   // SW_SQTS[11] := 8;
   // SW_SQTS[12] := 9;
   // SW_SQTS[13] := 10;
   // SW_SQTS[14] := 11;
   // SW_SQTS[15] := 12;
   // SW_SQTS[16] := 12;
   // SW_SQTS[17] := 13;
   // SW_SQTS[18] := 13;
   // SW_SQTS[19] := 13;
   // SW_SQTS[20] := 13;
   // SW_SQTS[21] := 14;
   // SW_SQTS[22] := 15;
   // SW_SQTS[23] := 16;
   // SW_SQTS[24] := 17;
   // SW_SQTS[25] := 17;
   // SW_SQTS[26] := 18;
   // SW_SQTS[27] := 19;
   // SW_SQTS[28] := 20;
   // SW_SQTS[29] := 21;
   // SW_SQTS[30] := 22;
   // SW_SQTS[31] := 23;
   // TVX[0] := 16#1;
   // TTX[0] := 16#1;
   // TSX[0] := 16#1;
   // S00X[0] := 16#1;
   // SOFFX[0] := 16#1;
   // SONX[0] := 16#1;
   // SAX[0] := 16#1;
   // SERRX[0] := 16#1;
   // SMX[0] := 16#1;
   // S0X[0] := 16#1;
   // S1X[0] := 16#1;
   // LSTT[47] := 20;
   // LSTT[48] := 25;
   // LSTT[49] := 21;
   // ATAJ[46] := 46;
   // ATAJ[47] := 47;
   // ATAJ[48] := 48;
   // ATAJ[49] := 49;
   // ATAB[46] := 1;
   // ATAB[47] := 33;
   // ATAB[48] := 34;
   // ATAB[49] := 27;
   // PSTT[46] := 1;
   // PSTT[47] := 23;
   // PSTT[48] := 27;
   // PSTT[49] := 20;
   // NSTT[47] := 20;
   // NSTT[48] := 25;
   // NSTT[49] := 21;
BEGIN
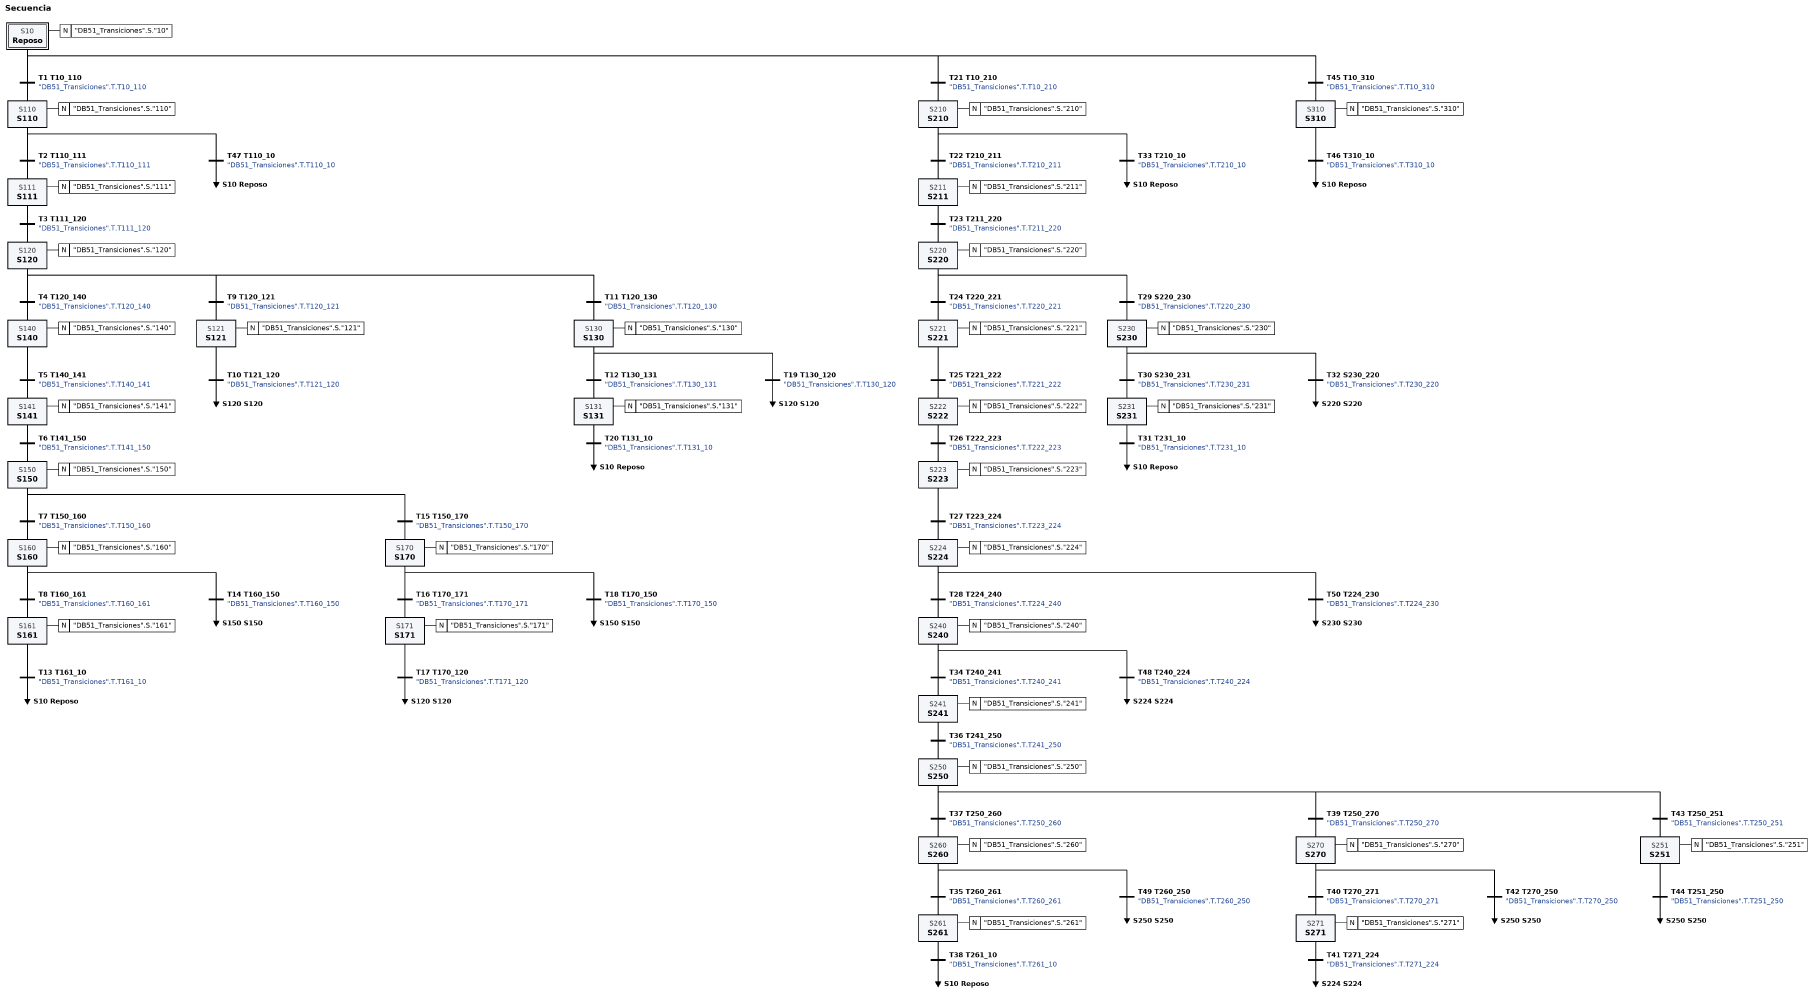
   // sequencer 1
   INITIAL_STEP Reposo:   // S10, max time T#10S, warning time T#7S
      // Estado inicial
              N    "DB51_Transiciones".S."10"
   END_STEP
   TRANSITION T10_110 FROM Reposo TO S110   // T1
      := "DB51_Transiciones".T.T10_110;
   END_TRANSITION
   TRANSITION T10_210 FROM Reposo TO S210   // T21
      := "DB51_Transiciones".T.T10_210;
   END_TRANSITION
   TRANSITION T10_310 FROM Reposo TO S310   // T45
      := "DB51_Transiciones".T.T10_310;
   END_TRANSITION
   STEP S110:   // S110, max time T#10S, warning time T#7S
      // Ingreso a bioterio: Solicitud ingreso Pasillo -> Vestuario
              N    "DB51_Transiciones".S."110"
   END_STEP
   TRANSITION T110_111 FROM S110 TO S111   // T2
      := "DB51_Transiciones".T.T110_111;
   END_TRANSITION
   TRANSITION T110_10 FROM S110 TO Reposo   // T47, jump
      := "DB51_Transiciones".T.T110_10;
   END_TRANSITION
   STEP S111:   // S111, max time T#10S, warning time T#7S
      // Ingreso a bioterio: Puerta P2-6 abierta
              N    "DB51_Transiciones".S."111"
   END_STEP
   TRANSITION T111_120 FROM S111 TO S120   // T3
      := "DB51_Transiciones".T.T111_120;
   END_TRANSITION
   STEP S120:   // S120, max time T#10S, warning time T#7S
      // Ingreso a bioterio: Vestuario ocupado
              N    "DB51_Transiciones".S."120"
   END_STEP
   TRANSITION T120_140 FROM S120 TO S140   // T4
      := "DB51_Transiciones".T.T120_140;
   END_TRANSITION
   TRANSITION T120_121 FROM S120 TO S121   // T9
      := "DB51_Transiciones".T.T120_121;
   END_TRANSITION
   TRANSITION T120_130 FROM S120 TO S130   // T11
      := "DB51_Transiciones".T.T120_130;
   END_TRANSITION
   STEP S140:   // S140, max time T#10S, warning time T#7S
      // Ingreso a bioterio: Solicitud ingreso Vestuario -> Ducha
              N    "DB51_Transiciones".S."140"
   END_STEP
   TRANSITION T140_141 FROM S140 TO S141   // T5
      := "DB51_Transiciones".T.T140_141;
   END_TRANSITION
   STEP S141:   // S141, max time T#10S, warning time T#7S
      // Ingreso a bioterio: Puerta P2-5 abierta
              N    "DB51_Transiciones".S."141"
   END_STEP
   TRANSITION T141_150 FROM S141 TO S150   // T6
      := "DB51_Transiciones".T.T141_150;
   END_TRANSITION
   STEP S150:   // S150, max time T#10S, warning time T#7S
      // Ingreso a bioterio: Ducha ocupada
              N    "DB51_Transiciones".S."150"
   END_STEP
   TRANSITION T150_160 FROM S150 TO S160   // T7
      := "DB51_Transiciones".T.T150_160;
   END_TRANSITION
   TRANSITION T150_170 FROM S150 TO S170   // T15
      := "DB51_Transiciones".T.T150_170;
   END_TRANSITION
   STEP S160:   // S160, max time T#10S, warning time T#7S
      // Ingreso a bioterio: Solicitud salir Ducha -> Bioterio
              N    "DB51_Transiciones".S."160"
   END_STEP
   TRANSITION T160_161 FROM S160 TO S161   // T8
      := "DB51_Transiciones".T.T160_161;
   END_TRANSITION
   TRANSITION T160_150 FROM S160 TO S150   // T14, jump
      := "DB51_Transiciones".T.T160_150;
   END_TRANSITION
   STEP S121:   // S121, max time T#10S, warning time T#7S
      // Ingreso a bioterio: Solicitud de precalentar ducha
              N    "DB51_Transiciones".S."121"
   END_STEP
   TRANSITION T121_120 FROM S121 TO S120   // T10, jump
      := "DB51_Transiciones".T.T121_120;
   END_TRANSITION
   STEP S130:   // S130, max time T#10S, warning time T#7S
      // Ingreso a bioterio: Solicitud salir Vestuario -> Pasillo
              N    "DB51_Transiciones".S."130"
   END_STEP
   TRANSITION T130_131 FROM S130 TO S131   // T12
      := "DB51_Transiciones".T.T130_131;
   END_TRANSITION
   TRANSITION T130_120 FROM S130 TO S120   // T19, jump
      := "DB51_Transiciones".T.T130_120;
   END_TRANSITION
   STEP S131:   // S131, max time T#10S, warning time T#7S
      // Ingreso a bioterio: Puerta P2-6 abierta
              N    "DB51_Transiciones".S."131"
   END_STEP
   TRANSITION T131_10 FROM S131 TO Reposo   // T20, jump
      := "DB51_Transiciones".T.T131_10;
   END_TRANSITION
   STEP S161:   // S161, max time T#10S, warning time T#7S
      // Ingreso a bioterio: Puerta P2-4 abierta
              N    "DB51_Transiciones".S."161"
   END_STEP
   TRANSITION T161_10 FROM S161 TO Reposo   // T13, jump
      := "DB51_Transiciones".T.T161_10;
   END_TRANSITION
   STEP S170:   // S170, max time T#10S, warning time T#7S
      // Ingreso a bioterio: Solicitud salir Ducha -> Vestuario
              N    "DB51_Transiciones".S."170"
   END_STEP
   TRANSITION T170_171 FROM S170 TO S171   // T16
      := "DB51_Transiciones".T.T170_171;
   END_TRANSITION
   TRANSITION T170_150 FROM S170 TO S150   // T18, jump
      := "DB51_Transiciones".T.T170_150;
   END_TRANSITION
   STEP S171:   // S171, max time T#10S, warning time T#7S
      // Ingreso a bioterio: Puerta P2-5 abierta
              N    "DB51_Transiciones".S."171"
   END_STEP
   TRANSITION T170_120 FROM S171 TO S120   // T17, jump
      := "DB51_Transiciones".T.T171_120;
   END_TRANSITION
   STEP S210:   // S210, max time T#10S, warning time T#7S
      // Egreso de bioterio: Solicitud ingreso Bioterio -> Ducha
              N    "DB51_Transiciones".S."210"
   END_STEP
   TRANSITION T210_211 FROM S210 TO S211   // T22
      := "DB51_Transiciones".T.T210_211;
   END_TRANSITION
   TRANSITION T210_10 FROM S210 TO Reposo   // T33, jump
      := "DB51_Transiciones".T.T210_10;
   END_TRANSITION
   STEP S211:   // S211, max time T#10S, warning time T#7S
      // Egreso de bioterio: Puerta P2-4 abierta
              N    "DB51_Transiciones".S."211"
   END_STEP
   TRANSITION T211_220 FROM S211 TO S220   // T23
      := "DB51_Transiciones".T.T211_220;
   END_TRANSITION
   STEP S220:   // S220, max time T#10S, warning time T#7S
      // Egreso de bioterio: Ducha ocupada - Espera incial
              N    "DB51_Transiciones".S."220"
   END_STEP
   TRANSITION T220_221 FROM S220 TO S221   // T24
      := "DB51_Transiciones".T.T220_221;
   END_TRANSITION
   TRANSITION S220_230 FROM S220 TO S230   // T29
      := "DB51_Transiciones".T.T220_230;
   END_TRANSITION
   STEP S221:   // S221, max time T#10S, warning time T#7S
      // Egreso de bioterio: Ducha ocupada - Válvula abierta
              N    "DB51_Transiciones".S."221"
   END_STEP
   TRANSITION T221_222 FROM S221 TO S222   // T25
      := "DB51_Transiciones".T.T221_222;
   END_TRANSITION
   STEP S222:   // S222, max time T#10S, warning time T#7S
      // Egreso de bioterio: Ducha ocupada - Pausa ducha
              N    "DB51_Transiciones".S."222"
   END_STEP
   TRANSITION T222_223 FROM S222 TO S223   // T26
      := "DB51_Transiciones".T.T222_223;
   END_TRANSITION
   STEP S223:   // S223, max time T#10S, warning time T#7S
      // Egreso de bioterio: Ducha ocupada - Válvula abierta
              N    "DB51_Transiciones".S."223"
   END_STEP
   TRANSITION T223_224 FROM S223 TO S224   // T27
      := "DB51_Transiciones".T.T223_224;
   END_TRANSITION
   STEP S224:   // S224, max time T#10S, warning time T#7S
      // Egreso de bioterio: Ducha ocupada
              N    "DB51_Transiciones".S."224"
   END_STEP
   TRANSITION T224_240 FROM S224 TO S240   // T28
      := "DB51_Transiciones".T.T224_240;
   END_TRANSITION
   TRANSITION T224_230 FROM S224 TO S230   // T50, jump
      := "DB51_Transiciones".T.T224_230;
   END_TRANSITION
   STEP S230:   // S230, max time T#10S, warning time T#7S
      // Egreso de bioterio: Solicitud salir Ducha -> Bioterio
              N    "DB51_Transiciones".S."230"
   END_STEP
   TRANSITION S230_231 FROM S230 TO S231   // T30
      := "DB51_Transiciones".T.T230_231;
   END_TRANSITION
   TRANSITION S230_220 FROM S230 TO S220   // T32, jump
      := "DB51_Transiciones".T.T230_220;
   END_TRANSITION
   STEP S231:   // S231, max time T#10S, warning time T#7S
      // Egreso de bioterio: Puerta P2-4 abierta
              N    "DB51_Transiciones".S."231"
   END_STEP
   TRANSITION T231_10 FROM S231 TO Reposo   // T31, jump
      := "DB51_Transiciones".T.T231_10;
   END_TRANSITION
   STEP S240:   // S240, max time T#10S, warning time T#7S
      // Egreso de bioterio: Solicitud salir Ducha -> Vestuario
              N    "DB51_Transiciones".S."240"
   END_STEP
   TRANSITION T240_241 FROM S240 TO S241   // T34
      := "DB51_Transiciones".T.T240_241;
   END_TRANSITION
   TRANSITION T240_224 FROM S240 TO S224   // T48, jump
      := "DB51_Transiciones".T.T240_224;
   END_TRANSITION
   STEP S241:   // S241, max time T#10S, warning time T#7S
      // Egreso de bioterio: Puerta P2-5 abierta
              N    "DB51_Transiciones".S."241"
   END_STEP
   TRANSITION T241_250 FROM S241 TO S250   // T36
      := "DB51_Transiciones".T.T241_250;
   END_TRANSITION
   STEP S250:   // S250, max time T#10S, warning time T#7S
      // Egreso de bioterio: Vestuario ocupado
              N    "DB51_Transiciones".S."250"
   END_STEP
   TRANSITION T250_260 FROM S250 TO S260   // T37
      := "DB51_Transiciones".T.T250_260;
   END_TRANSITION
   TRANSITION T250_270 FROM S250 TO S270   // T39
      := "DB51_Transiciones".T.T250_270;
   END_TRANSITION
   TRANSITION T250_251 FROM S250 TO S251   // T43
      := "DB51_Transiciones".T.T250_251;
   END_TRANSITION
   STEP S260:   // S260, max time T#10S, warning time T#7S
      // Egreso de bioterio: Solicitud salir Vestuario -> Pasillo
              N    "DB51_Transiciones".S."260"
   END_STEP
   TRANSITION T260_261 FROM S260 TO S261   // T35
      := "DB51_Transiciones".T.T260_261;
   END_TRANSITION
   TRANSITION T260_250 FROM S260 TO S250   // T49, jump
      := "DB51_Transiciones".T.T260_250;
   END_TRANSITION
   STEP S261:   // S261, max time T#10S, warning time T#7S
      // Egreso de bioterio: Puerta P2-6 abierta
              N    "DB51_Transiciones".S."261"
   END_STEP
   TRANSITION T261_10 FROM S261 TO Reposo   // T38, jump
      := "DB51_Transiciones".T.T261_10;
   END_TRANSITION
   STEP S270:   // S270, max time T#10S, warning time T#7S
      // Egreso de bioterio: Solicitud ingreso Vestuario -> Ducha
              N    "DB51_Transiciones".S."270"
   END_STEP
   TRANSITION T270_271 FROM S270 TO S271   // T40
      := "DB51_Transiciones".T.T270_271;
   END_TRANSITION
   TRANSITION T270_250 FROM S270 TO S250   // T42, jump
      := "DB51_Transiciones".T.T270_250;
   END_TRANSITION
   STEP S271:   // S271, max time T#10S, warning time T#7S
      // Egreso de bioterio: Puerta P2-5 abierta
              N    "DB51_Transiciones".S."271"
   END_STEP
   TRANSITION T271_224 FROM S271 TO S224   // T41, jump
      := "DB51_Transiciones".T.T271_224;
   END_TRANSITION
   STEP S251:   // S251, max time T#10S, warning time T#7S
      // Egreso de bioterio: Solicitud de precalentar ducha
              N    "DB51_Transiciones".S."251"
   END_STEP
   TRANSITION T251_250 FROM S251 TO S250   // T44, jump
      := "DB51_Transiciones".T.T251_250;
   END_TRANSITION
   STEP S310:   // S310, max time T#10S, warning time T#7S
      // Egreso de bioterio: Solicitud de precalentar ducha
              N    "DB51_Transiciones".S."310"
   END_STEP
   TRANSITION T310_10 FROM S310 TO Reposo   // T46, jump
      := "DB51_Transiciones".T.T310_10;
   END_TRANSITION
END_FUNCTION_BLOCK

FUNCTION "COM_SCADA" : Void   // FC1, LAD
TITLE = Comunicación con SCADA
{ S7_Optimized_Access := 'TRUE' }
VERSION : 0.1
BEGIN

REGION Network 1: Comunicación con SCADA
END_REGION

REGION Network 2: DATOS SCADA -> PLC
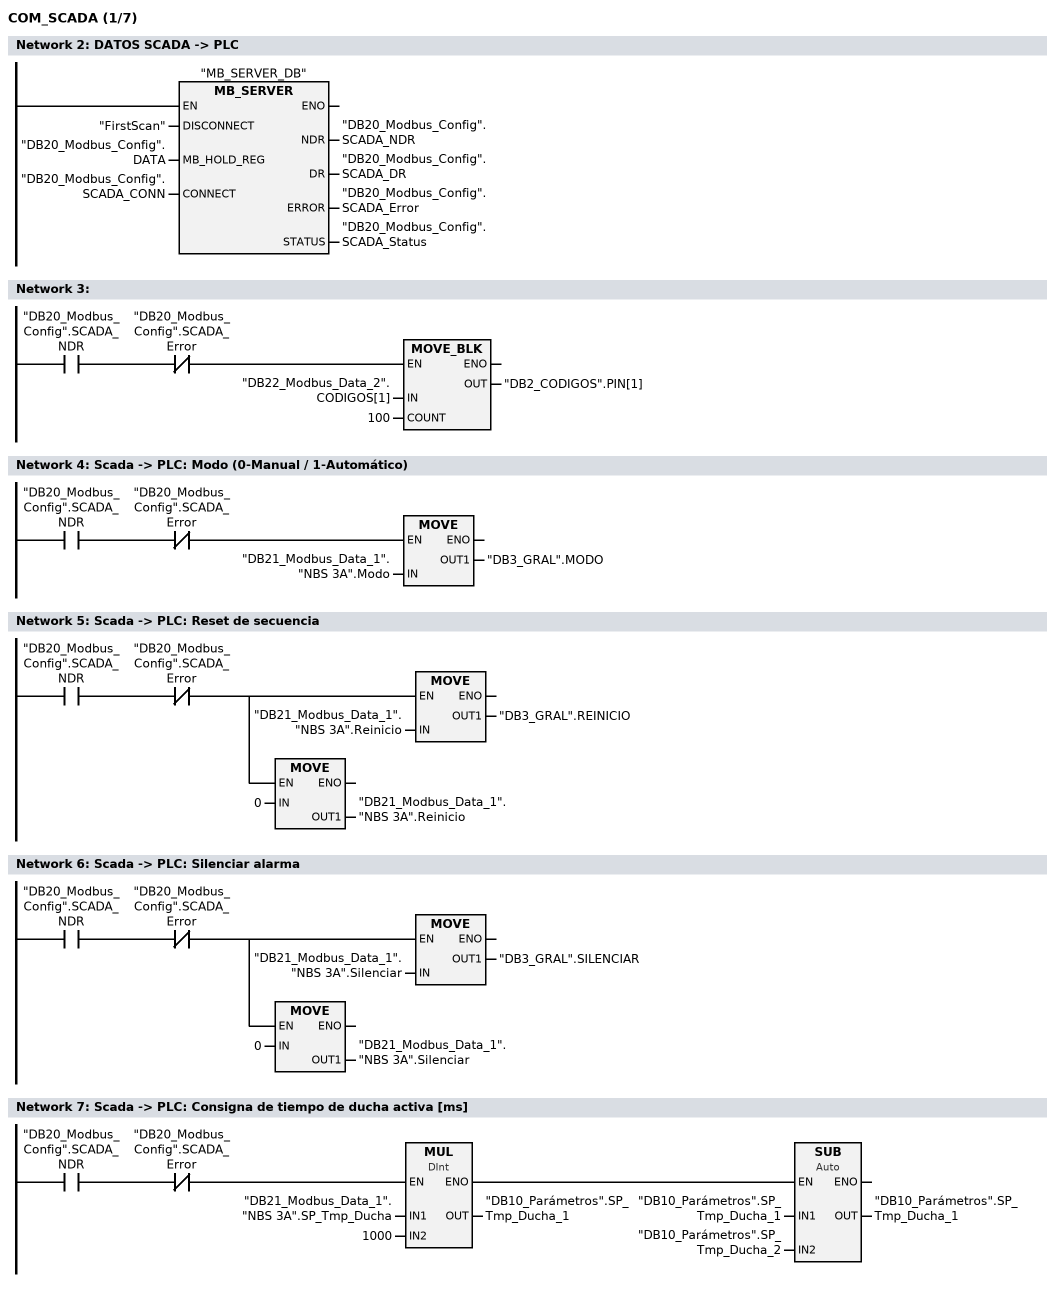
   "MB_SERVER_DB"(DISCONNECT := "FirstScan",   // MB_SERVER
                  MB_HOLD_REG := "DB20_Modbus_Config".DATA,
                  CONNECT := "DB20_Modbus_Config".SCADA_CONN,
                  NDR => "DB20_Modbus_Config".SCADA_NDR,
                  DR => "DB20_Modbus_Config".SCADA_DR,
                  ERROR => "DB20_Modbus_Config".SCADA_Error,
                  STATUS => "DB20_Modbus_Config".SCADA_Status);
END_REGION

REGION Network 3
   IF "DB20_Modbus_Config".SCADA_NDR AND NOT "DB20_Modbus_Config".SCADA_Error THEN
       MOVE_BLK(IN := "DB22_Modbus_Data_2".CODIGOS[1], COUNT := 100, OUT => "DB2_CODIGOS".PIN[1]);
   END_IF;
END_REGION

REGION Network 4: Scada -> PLC: Modo (0-Manual / 1-Automático)
   RUNG wire#powerrail
      Contact( "DB20_Modbus_Config".SCADA_NDR )
      I_Contact( "DB20_Modbus_Config".SCADA_Error )
      Move(in := "DB21_Modbus_Data_1"."NBS 3A".Modo, out1 => "DB3_GRAL".MODO)
   END_RUNG
   // the same network as SCL:
   IF "DB20_Modbus_Config".SCADA_NDR AND NOT "DB20_Modbus_Config".SCADA_Error THEN
       "DB3_GRAL".MODO := "DB21_Modbus_Data_1"."NBS 3A".Modo;
   END_IF;
END_REGION

REGION Network 5: Scada -> PLC: Reset de secuencia
   RUNG wire#powerrail
      Contact( "DB20_Modbus_Config".SCADA_NDR )
      I_Contact( "DB20_Modbus_Config".SCADA_Error )
      wire#w1
      Move(in := "DB21_Modbus_Data_1"."NBS 3A".Reinicio, out1 => "DB3_GRAL".REINICIO)
   END_RUNG
   RUNG wire#w1
      Move(in := 0, out1 => "DB21_Modbus_Data_1"."NBS 3A".Reinicio)
   END_RUNG
   // the same network as SCL:
   IF "DB20_Modbus_Config".SCADA_NDR AND NOT "DB20_Modbus_Config".SCADA_Error THEN
       "DB3_GRAL".REINICIO := "DB21_Modbus_Data_1"."NBS 3A".Reinicio;
       "DB21_Modbus_Data_1"."NBS 3A".Reinicio := 0;
   END_IF;
END_REGION

REGION Network 6: Scada -> PLC: Silenciar alarma
   RUNG wire#powerrail
      Contact( "DB20_Modbus_Config".SCADA_NDR )
      I_Contact( "DB20_Modbus_Config".SCADA_Error )
      wire#w1
      Move(in := "DB21_Modbus_Data_1"."NBS 3A".Silenciar, out1 => "DB3_GRAL".SILENCIAR)
   END_RUNG
   RUNG wire#w1
      Move(in := 0, out1 => "DB21_Modbus_Data_1"."NBS 3A".Silenciar)
   END_RUNG
   // the same network as SCL:
   IF "DB20_Modbus_Config".SCADA_NDR AND NOT "DB20_Modbus_Config".SCADA_Error THEN
       "DB3_GRAL".SILENCIAR := "DB21_Modbus_Data_1"."NBS 3A".Silenciar;
       "DB21_Modbus_Data_1"."NBS 3A".Silenciar := 0;
   END_IF;
END_REGION

REGION Network 7: Scada -> PLC: Consigna de tiempo de ducha activa [ms]
   RUNG wire#powerrail
      Contact( "DB20_Modbus_Config".SCADA_NDR )
      I_Contact( "DB20_Modbus_Config".SCADA_Error )
      { S7_Templates := "SrcType := DInt" } Mul(in1 := "DB21_Modbus_Data_1"."NBS 3A".SP_Tmp_Ducha, in2 := 1000, out => "DB10_Parámetros".SP_Tmp_Ducha_1)
      Sub(in1 := "DB10_Parámetros".SP_Tmp_Ducha_1, in2 := "DB10_Parámetros".SP_Tmp_Ducha_2, out => "DB10_Parámetros".SP_Tmp_Ducha_1)
   END_RUNG
   // the same network as SCL:
   IF "DB20_Modbus_Config".SCADA_NDR AND NOT "DB20_Modbus_Config".SCADA_Error THEN
       "DB10_Parámetros".SP_Tmp_Ducha_1 := "DB21_Modbus_Data_1"."NBS 3A".SP_Tmp_Ducha * 1000;
       "DB10_Parámetros".SP_Tmp_Ducha_1 := "DB10_Parámetros".SP_Tmp_Ducha_1 - "DB10_Parámetros".SP_Tmp_Ducha_2;
   END_IF;
END_REGION

REGION Network 8: Scada -> PLC: Consigna de tiempo de precalentar ducha [ms]
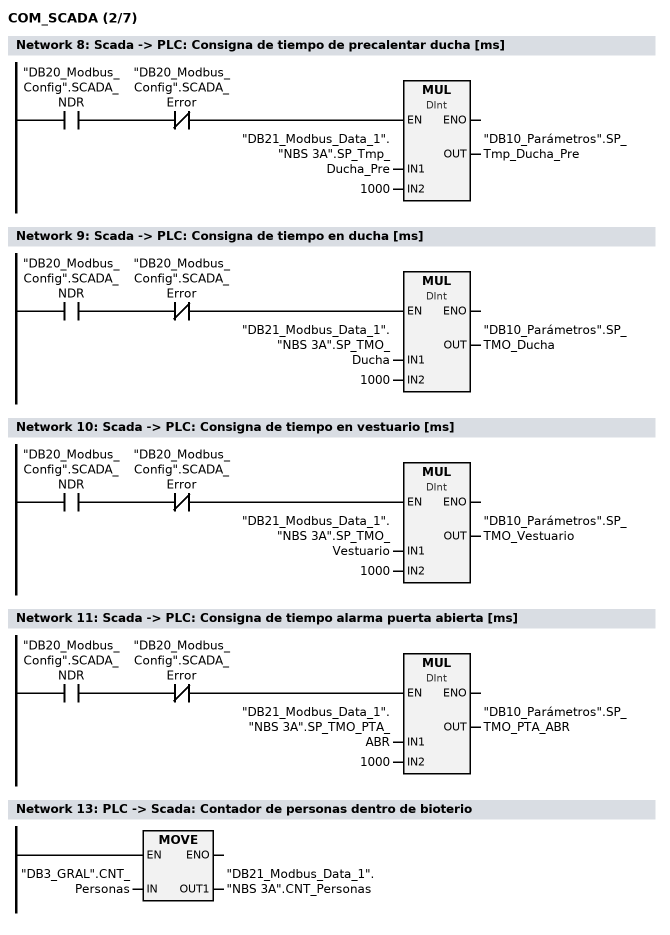
   RUNG wire#powerrail
      Contact( "DB20_Modbus_Config".SCADA_NDR )
      I_Contact( "DB20_Modbus_Config".SCADA_Error )
      { S7_Templates := "SrcType := DInt" } Mul(in1 := "DB21_Modbus_Data_1"."NBS 3A".SP_Tmp_Ducha_Pre, in2 := 1000, out => "DB10_Parámetros".SP_Tmp_Ducha_Pre)
   END_RUNG
   // the same network as SCL:
   IF "DB20_Modbus_Config".SCADA_NDR AND NOT "DB20_Modbus_Config".SCADA_Error THEN
       "DB10_Parámetros".SP_Tmp_Ducha_Pre := "DB21_Modbus_Data_1"."NBS 3A".SP_Tmp_Ducha_Pre * 1000;
   END_IF;
END_REGION

REGION Network 9: Scada -> PLC: Consigna de tiempo en ducha [ms]
   RUNG wire#powerrail
      Contact( "DB20_Modbus_Config".SCADA_NDR )
      I_Contact( "DB20_Modbus_Config".SCADA_Error )
      { S7_Templates := "SrcType := DInt" } Mul(in1 := "DB21_Modbus_Data_1"."NBS 3A".SP_TMO_Ducha, in2 := 1000, out => "DB10_Parámetros".SP_TMO_Ducha)
   END_RUNG
   // the same network as SCL:
   IF "DB20_Modbus_Config".SCADA_NDR AND NOT "DB20_Modbus_Config".SCADA_Error THEN
       "DB10_Parámetros".SP_TMO_Ducha := "DB21_Modbus_Data_1"."NBS 3A".SP_TMO_Ducha * 1000;
   END_IF;
END_REGION

REGION Network 10: Scada -> PLC: Consigna de tiempo en vestuario [ms]
   RUNG wire#powerrail
      Contact( "DB20_Modbus_Config".SCADA_NDR )
      I_Contact( "DB20_Modbus_Config".SCADA_Error )
      { S7_Templates := "SrcType := DInt" } Mul(in1 := "DB21_Modbus_Data_1"."NBS 3A".SP_TMO_Vestuario, in2 := 1000, out => "DB10_Parámetros".SP_TMO_Vestuario)
   END_RUNG
   // the same network as SCL:
   IF "DB20_Modbus_Config".SCADA_NDR AND NOT "DB20_Modbus_Config".SCADA_Error THEN
       "DB10_Parámetros".SP_TMO_Vestuario := "DB21_Modbus_Data_1"."NBS 3A".SP_TMO_Vestuario * 1000;
   END_IF;
END_REGION

REGION Network 11: Scada -> PLC: Consigna de tiempo alarma puerta abierta [ms]
   RUNG wire#powerrail
      Contact( "DB20_Modbus_Config".SCADA_NDR )
      I_Contact( "DB20_Modbus_Config".SCADA_Error )
      { S7_Templates := "SrcType := DInt" } Mul(in1 := "DB21_Modbus_Data_1"."NBS 3A".SP_TMO_PTA_ABR, in2 := 1000, out => "DB10_Parámetros".SP_TMO_PTA_ABR)
   END_RUNG
   // the same network as SCL:
   IF "DB20_Modbus_Config".SCADA_NDR AND NOT "DB20_Modbus_Config".SCADA_Error THEN
       "DB10_Parámetros".SP_TMO_PTA_ABR := "DB21_Modbus_Data_1"."NBS 3A".SP_TMO_PTA_ABR * 1000;
   END_IF;
END_REGION

REGION Network 12: DATOS PLC -> SCADA
END_REGION

REGION Network 13: PLC -> Scada: Contador de personas dentro de bioterio
   RUNG wire#powerrail
      Move(in := "DB3_GRAL".CNT_Personas, out1 => "DB21_Modbus_Data_1"."NBS 3A".CNT_Personas)
   END_RUNG
   // the same network as SCL:
   "DB21_Modbus_Data_1"."NBS 3A".CNT_Personas := "DB3_GRAL".CNT_Personas;
END_REGION

REGION Network 14: PLC -> Scada: P2-6 - Puerta Pasillo: Estado (0-Cerrada / 1-Abierta / 2-Falla reconocida / 3-Falla nueva)
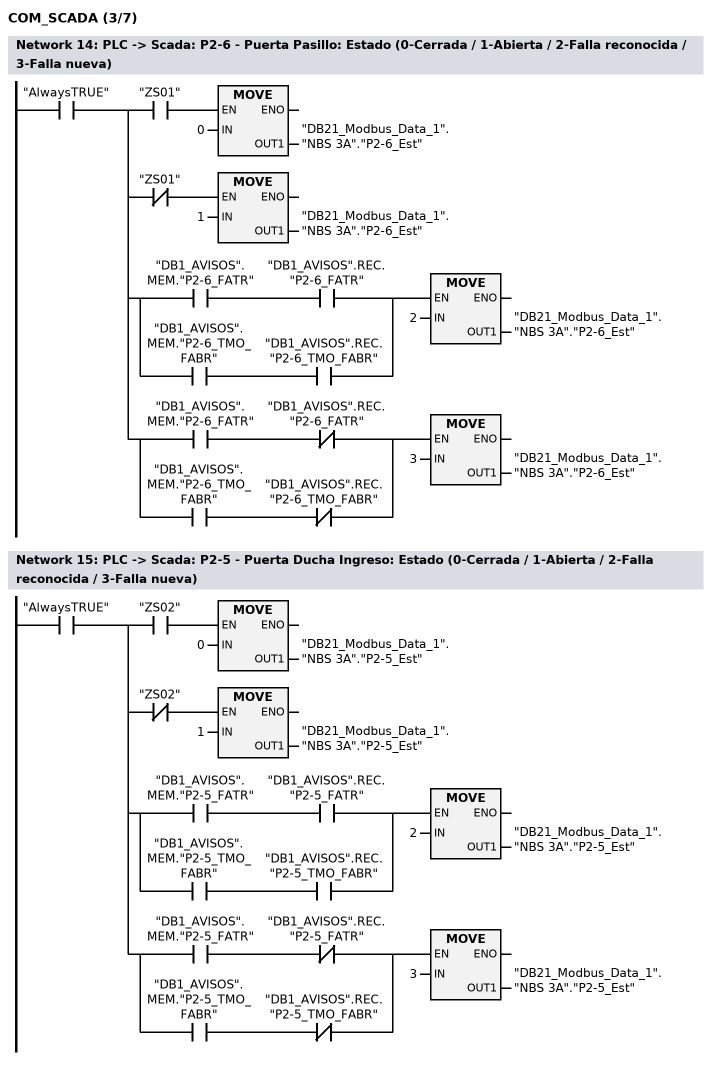
   RUNG wire#powerrail
      Contact( "AlwaysTRUE" )
      wire#w1
      Contact( "ZS01" )
      Move(in := 0, out1 => "DB21_Modbus_Data_1"."NBS 3A"."P2-6_Est")
   END_RUNG
   RUNG wire#w1
      I_Contact( "ZS01" )
      Move(in := 1, out1 => "DB21_Modbus_Data_1"."NBS 3A"."P2-6_Est")
   END_RUNG
   RUNG wire#w1
      Contact( "DB1_AVISOS".MEM."P2-6_FATR" )
      Contact( "DB1_AVISOS".REC."P2-6_FATR" )
      wire#w2
      Move(in := 2, out1 => "DB21_Modbus_Data_1"."NBS 3A"."P2-6_Est")
   END_RUNG
   RUNG wire#w1
      Contact( "DB1_AVISOS".MEM."P2-6_TMO_FABR" )
      Contact( "DB1_AVISOS".REC."P2-6_TMO_FABR" )
   END_RUNG wire#w2
   RUNG wire#w1
      Contact( "DB1_AVISOS".MEM."P2-6_FATR" )
      I_Contact( "DB1_AVISOS".REC."P2-6_FATR" )
      wire#w3
      Move(in := 3, out1 => "DB21_Modbus_Data_1"."NBS 3A"."P2-6_Est")
   END_RUNG
   RUNG wire#w1
      Contact( "DB1_AVISOS".MEM."P2-6_TMO_FABR" )
      I_Contact( "DB1_AVISOS".REC."P2-6_TMO_FABR" )
   END_RUNG wire#w3
   // the same network as SCL:
   IF "AlwaysTRUE" AND "ZS01" THEN "DB21_Modbus_Data_1"."NBS 3A"."P2-6_Est" := 0; END_IF;
   IF "AlwaysTRUE" AND NOT "ZS01" THEN "DB21_Modbus_Data_1"."NBS 3A"."P2-6_Est" := 1; END_IF;
   IF "AlwaysTRUE" AND (("DB1_AVISOS".MEM."P2-6_FATR" AND "DB1_AVISOS".REC."P2-6_FATR") OR ("DB1_AVISOS".MEM."P2-6_TMO_FABR" AND "DB1_AVISOS".REC."P2-6_TMO_FABR")) THEN
       "DB21_Modbus_Data_1"."NBS 3A"."P2-6_Est" := 2;
   END_IF;
   IF "AlwaysTRUE" AND (("DB1_AVISOS".MEM."P2-6_FATR" AND NOT "DB1_AVISOS".REC."P2-6_FATR") OR ("DB1_AVISOS".MEM."P2-6_TMO_FABR" AND NOT "DB1_AVISOS".REC."P2-6_TMO_FABR")) THEN
       "DB21_Modbus_Data_1"."NBS 3A"."P2-6_Est" := 3;
   END_IF;
END_REGION

REGION Network 15: PLC -> Scada: P2-5 - Puerta Ducha Ingreso: Estado (0-Cerrada / 1-Abierta / 2-Falla reconocida / 3-Falla nueva)
   RUNG wire#powerrail
      Contact( "AlwaysTRUE" )
      wire#w1
      Contact( "ZS02" )
      Move(in := 0, out1 => "DB21_Modbus_Data_1"."NBS 3A"."P2-5_Est")
   END_RUNG
   RUNG wire#w1
      I_Contact( "ZS02" )
      Move(in := 1, out1 => "DB21_Modbus_Data_1"."NBS 3A"."P2-5_Est")
   END_RUNG
   RUNG wire#w1
      Contact( "DB1_AVISOS".MEM."P2-5_FATR" )
      Contact( "DB1_AVISOS".REC."P2-5_FATR" )
      wire#w2
      Move(in := 2, out1 => "DB21_Modbus_Data_1"."NBS 3A"."P2-5_Est")
   END_RUNG
   RUNG wire#w1
      Contact( "DB1_AVISOS".MEM."P2-5_TMO_FABR" )
      Contact( "DB1_AVISOS".REC."P2-5_TMO_FABR" )
   END_RUNG wire#w2
   RUNG wire#w1
      Contact( "DB1_AVISOS".MEM."P2-5_FATR" )
      I_Contact( "DB1_AVISOS".REC."P2-5_FATR" )
      wire#w3
      Move(in := 3, out1 => "DB21_Modbus_Data_1"."NBS 3A"."P2-5_Est")
   END_RUNG
   RUNG wire#w1
      Contact( "DB1_AVISOS".MEM."P2-5_TMO_FABR" )
      I_Contact( "DB1_AVISOS".REC."P2-5_TMO_FABR" )
   END_RUNG wire#w3
   // the same network as SCL:
   IF "AlwaysTRUE" AND "ZS02" THEN "DB21_Modbus_Data_1"."NBS 3A"."P2-5_Est" := 0; END_IF;
   IF "AlwaysTRUE" AND NOT "ZS02" THEN "DB21_Modbus_Data_1"."NBS 3A"."P2-5_Est" := 1; END_IF;
   IF "AlwaysTRUE" AND (("DB1_AVISOS".MEM."P2-5_FATR" AND "DB1_AVISOS".REC."P2-5_FATR") OR ("DB1_AVISOS".MEM."P2-5_TMO_FABR" AND "DB1_AVISOS".REC."P2-5_TMO_FABR")) THEN
       "DB21_Modbus_Data_1"."NBS 3A"."P2-5_Est" := 2;
   END_IF;
   IF "AlwaysTRUE" AND (("DB1_AVISOS".MEM."P2-5_FATR" AND NOT "DB1_AVISOS".REC."P2-5_FATR") OR ("DB1_AVISOS".MEM."P2-5_TMO_FABR" AND NOT "DB1_AVISOS".REC."P2-5_TMO_FABR")) THEN
       "DB21_Modbus_Data_1"."NBS 3A"."P2-5_Est" := 3;
   END_IF;
END_REGION

REGION Network 16: PLC -> Scada: P2-4 - Puerta Ducha Salida: Estado (0-Cerrada / 1-Abierta / 2-Falla reconocida / 3-Falla nueva)
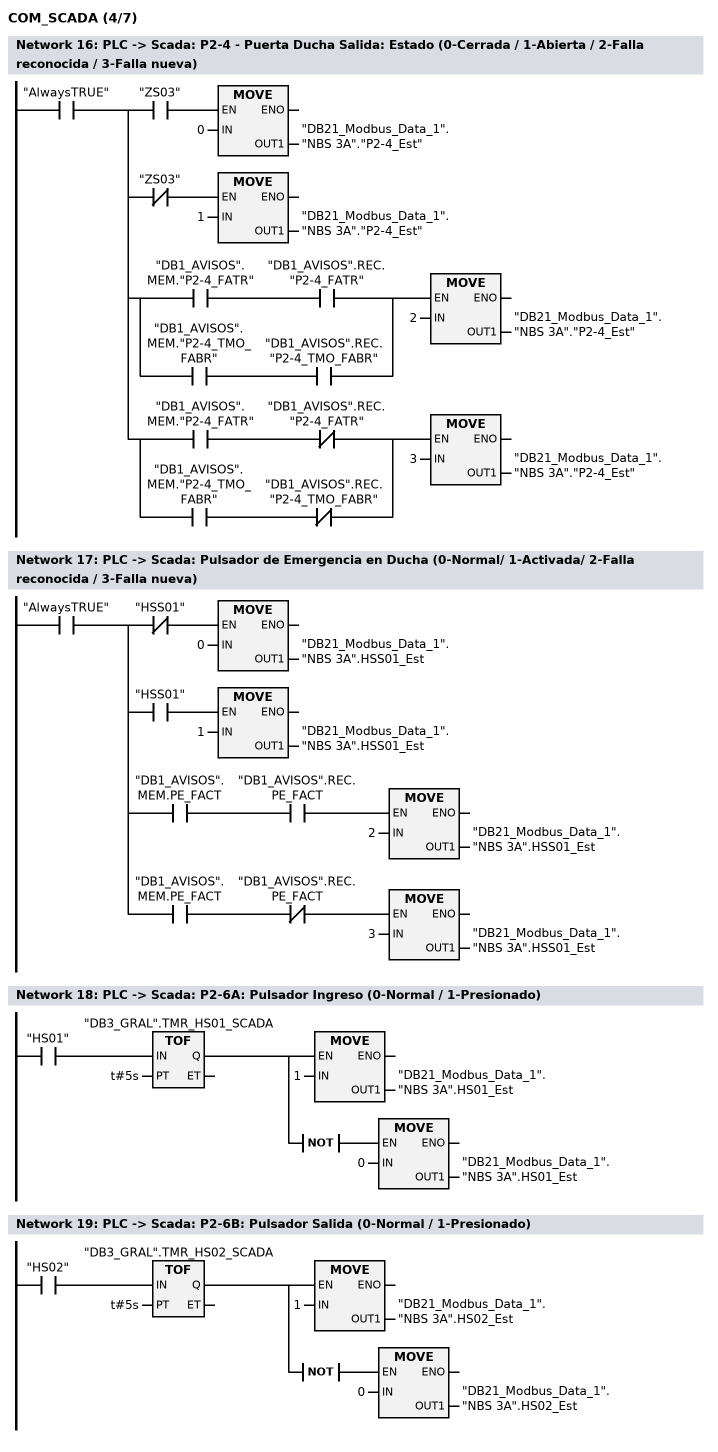
   RUNG wire#powerrail
      Contact( "AlwaysTRUE" )
      wire#w1
      Contact( "ZS03" )
      Move(in := 0, out1 => "DB21_Modbus_Data_1"."NBS 3A"."P2-4_Est")
   END_RUNG
   RUNG wire#w1
      I_Contact( "ZS03" )
      Move(in := 1, out1 => "DB21_Modbus_Data_1"."NBS 3A"."P2-4_Est")
   END_RUNG
   RUNG wire#w1
      Contact( "DB1_AVISOS".MEM."P2-4_FATR" )
      Contact( "DB1_AVISOS".REC."P2-4_FATR" )
      wire#w2
      Move(in := 2, out1 => "DB21_Modbus_Data_1"."NBS 3A"."P2-4_Est")
   END_RUNG
   RUNG wire#w1
      Contact( "DB1_AVISOS".MEM."P2-4_TMO_FABR" )
      Contact( "DB1_AVISOS".REC."P2-4_TMO_FABR" )
   END_RUNG wire#w2
   RUNG wire#w1
      Contact( "DB1_AVISOS".MEM."P2-4_FATR" )
      I_Contact( "DB1_AVISOS".REC."P2-4_FATR" )
      wire#w3
      Move(in := 3, out1 => "DB21_Modbus_Data_1"."NBS 3A"."P2-4_Est")
   END_RUNG
   RUNG wire#w1
      Contact( "DB1_AVISOS".MEM."P2-4_TMO_FABR" )
      I_Contact( "DB1_AVISOS".REC."P2-4_TMO_FABR" )
   END_RUNG wire#w3
   // the same network as SCL:
   IF "AlwaysTRUE" AND "ZS03" THEN "DB21_Modbus_Data_1"."NBS 3A"."P2-4_Est" := 0; END_IF;
   IF "AlwaysTRUE" AND NOT "ZS03" THEN "DB21_Modbus_Data_1"."NBS 3A"."P2-4_Est" := 1; END_IF;
   IF "AlwaysTRUE" AND (("DB1_AVISOS".MEM."P2-4_FATR" AND "DB1_AVISOS".REC."P2-4_FATR") OR ("DB1_AVISOS".MEM."P2-4_TMO_FABR" AND "DB1_AVISOS".REC."P2-4_TMO_FABR")) THEN
       "DB21_Modbus_Data_1"."NBS 3A"."P2-4_Est" := 2;
   END_IF;
   IF "AlwaysTRUE" AND (("DB1_AVISOS".MEM."P2-4_FATR" AND NOT "DB1_AVISOS".REC."P2-4_FATR") OR ("DB1_AVISOS".MEM."P2-4_TMO_FABR" AND NOT "DB1_AVISOS".REC."P2-4_TMO_FABR")) THEN
       "DB21_Modbus_Data_1"."NBS 3A"."P2-4_Est" := 3;
   END_IF;
END_REGION

REGION Network 17: PLC -> Scada: Pulsador de Emergencia en Ducha (0-Normal/ 1-Activada/ 2-Falla reconocida / 3-Falla nueva)
   RUNG wire#powerrail
      Contact( "AlwaysTRUE" )
      wire#w1
      I_Contact( "HSS01" )
      Move(in := 0, out1 => "DB21_Modbus_Data_1"."NBS 3A".HSS01_Est)
   END_RUNG
   RUNG wire#w1
      Contact( "HSS01" )
      Move(in := 1, out1 => "DB21_Modbus_Data_1"."NBS 3A".HSS01_Est)
   END_RUNG
   RUNG wire#w1
      Contact( "DB1_AVISOS".MEM.PE_FACT )
      Contact( "DB1_AVISOS".REC.PE_FACT )
      Move(in := 2, out1 => "DB21_Modbus_Data_1"."NBS 3A".HSS01_Est)
   END_RUNG
   RUNG wire#w1
      Contact( "DB1_AVISOS".MEM.PE_FACT )
      I_Contact( "DB1_AVISOS".REC.PE_FACT )
      Move(in := 3, out1 => "DB21_Modbus_Data_1"."NBS 3A".HSS01_Est)
   END_RUNG
   // the same network as SCL:
   IF "AlwaysTRUE" AND NOT "HSS01" THEN "DB21_Modbus_Data_1"."NBS 3A".HSS01_Est := 0; END_IF;
   IF "AlwaysTRUE" AND "HSS01" THEN "DB21_Modbus_Data_1"."NBS 3A".HSS01_Est := 1; END_IF;
   IF "AlwaysTRUE" AND "DB1_AVISOS".MEM.PE_FACT AND "DB1_AVISOS".REC.PE_FACT THEN
       "DB21_Modbus_Data_1"."NBS 3A".HSS01_Est := 2;
   END_IF;
   IF "AlwaysTRUE" AND "DB1_AVISOS".MEM.PE_FACT AND NOT "DB1_AVISOS".REC.PE_FACT THEN
       "DB21_Modbus_Data_1"."NBS 3A".HSS01_Est := 3;
   END_IF;
END_REGION

REGION Network 18: PLC -> Scada: P2-6A: Pulsador Ingreso (0-Normal / 1-Presionado)
   "DB3_GRAL".TMR_HS01_SCADA.TOF(IN := "HS01", PT := t#5s);
   IF "DB3_GRAL".TMR_HS01_SCADA.Q THEN "DB21_Modbus_Data_1"."NBS 3A".HS01_Est := 1; END_IF;
   IF NOT "DB3_GRAL".TMR_HS01_SCADA.Q THEN "DB21_Modbus_Data_1"."NBS 3A".HS01_Est := 0; END_IF;
END_REGION

REGION Network 19: PLC -> Scada: P2-6B: Pulsador Salida (0-Normal / 1-Presionado)
   "DB3_GRAL".TMR_HS02_SCADA.TOF(IN := "HS02", PT := t#5s);
   IF "DB3_GRAL".TMR_HS02_SCADA.Q THEN "DB21_Modbus_Data_1"."NBS 3A".HS02_Est := 1; END_IF;
   IF NOT "DB3_GRAL".TMR_HS02_SCADA.Q THEN "DB21_Modbus_Data_1"."NBS 3A".HS02_Est := 0; END_IF;
END_REGION

REGION Network 20: PLC -> Scada: P2-5A: Pulsador Salida (0-Normal / 1-Presionado)
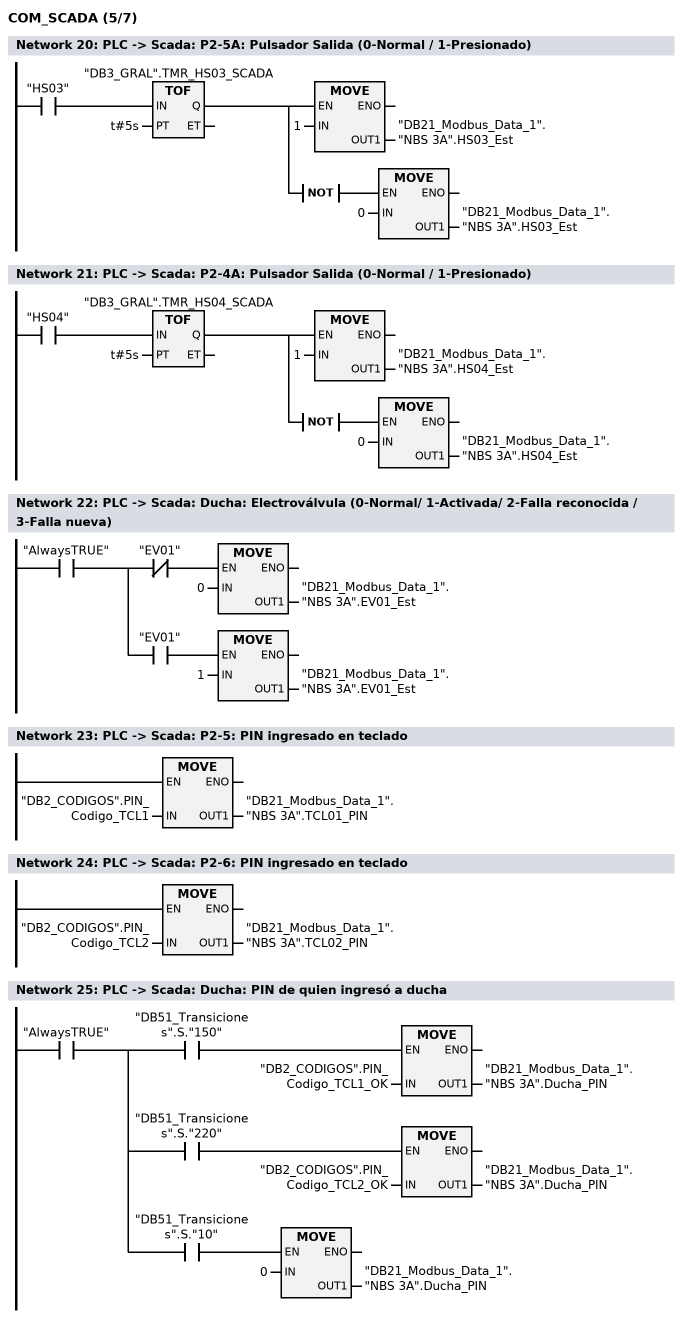
   "DB3_GRAL".TMR_HS03_SCADA.TOF(IN := "HS03", PT := t#5s);
   IF "DB3_GRAL".TMR_HS03_SCADA.Q THEN "DB21_Modbus_Data_1"."NBS 3A".HS03_Est := 1; END_IF;
   IF NOT "DB3_GRAL".TMR_HS03_SCADA.Q THEN "DB21_Modbus_Data_1"."NBS 3A".HS03_Est := 0; END_IF;
END_REGION

REGION Network 21: PLC -> Scada: P2-4A: Pulsador Salida (0-Normal / 1-Presionado)
   "DB3_GRAL".TMR_HS04_SCADA.TOF(IN := "HS04", PT := t#5s);
   IF "DB3_GRAL".TMR_HS04_SCADA.Q THEN "DB21_Modbus_Data_1"."NBS 3A".HS04_Est := 1; END_IF;
   IF NOT "DB3_GRAL".TMR_HS04_SCADA.Q THEN "DB21_Modbus_Data_1"."NBS 3A".HS04_Est := 0; END_IF;
END_REGION

REGION Network 22: PLC -> Scada: Ducha: Electroválvula (0-Normal/ 1-Activada/ 2-Falla reconocida / 3-Falla nueva)
   RUNG wire#powerrail
      Contact( "AlwaysTRUE" )
      wire#w1
      I_Contact( "EV01" )
      Move(in := 0, out1 => "DB21_Modbus_Data_1"."NBS 3A".EV01_Est)
   END_RUNG
   RUNG wire#w1
      Contact( "EV01" )
      Move(in := 1, out1 => "DB21_Modbus_Data_1"."NBS 3A".EV01_Est)
   END_RUNG
   // the same network as SCL:
   IF "AlwaysTRUE" AND NOT "EV01" THEN "DB21_Modbus_Data_1"."NBS 3A".EV01_Est := 0; END_IF;
   IF "AlwaysTRUE" AND "EV01" THEN "DB21_Modbus_Data_1"."NBS 3A".EV01_Est := 1; END_IF;
END_REGION

REGION Network 23: PLC -> Scada: P2-5: PIN ingresado en teclado
   RUNG wire#powerrail
      Move(in := "DB2_CODIGOS".PIN_Codigo_TCL1, out1 => "DB21_Modbus_Data_1"."NBS 3A".TCL01_PIN)
   END_RUNG
   // the same network as SCL:
   "DB21_Modbus_Data_1"."NBS 3A".TCL01_PIN := "DB2_CODIGOS".PIN_Codigo_TCL1;
END_REGION

REGION Network 24: PLC -> Scada: P2-6: PIN ingresado en teclado
   RUNG wire#powerrail
      Move(in := "DB2_CODIGOS".PIN_Codigo_TCL2, out1 => "DB21_Modbus_Data_1"."NBS 3A".TCL02_PIN)
   END_RUNG
   // the same network as SCL:
   "DB21_Modbus_Data_1"."NBS 3A".TCL02_PIN := "DB2_CODIGOS".PIN_Codigo_TCL2;
END_REGION

REGION Network 25: PLC -> Scada: Ducha: PIN de quien ingresó a ducha
   RUNG wire#powerrail
      Contact( "AlwaysTRUE" )
      wire#w1
      Contact( "DB51_Transiciones".S."150" )
      Move(in := "DB2_CODIGOS".PIN_Codigo_TCL1_OK, out1 => "DB21_Modbus_Data_1"."NBS 3A".Ducha_PIN)
   END_RUNG
   RUNG wire#w1
      Contact( "DB51_Transiciones".S."220" )
      Move(in := "DB2_CODIGOS".PIN_Codigo_TCL2_OK, out1 => "DB21_Modbus_Data_1"."NBS 3A".Ducha_PIN)
   END_RUNG
   RUNG wire#w1
      Contact( "DB51_Transiciones".S."10" )
      Move(in := 0, out1 => "DB21_Modbus_Data_1"."NBS 3A".Ducha_PIN)
   END_RUNG
   // the same network as SCL:
   IF "AlwaysTRUE" AND "DB51_Transiciones".S."150" THEN
       "DB21_Modbus_Data_1"."NBS 3A".Ducha_PIN := "DB2_CODIGOS".PIN_Codigo_TCL1_OK;
   END_IF;
   IF "AlwaysTRUE" AND "DB51_Transiciones".S."220" THEN
       "DB21_Modbus_Data_1"."NBS 3A".Ducha_PIN := "DB2_CODIGOS".PIN_Codigo_TCL2_OK;
   END_IF;
   IF "AlwaysTRUE" AND "DB51_Transiciones".S."10" THEN "DB21_Modbus_Data_1"."NBS 3A".Ducha_PIN := 0; END_IF;
END_REGION

REGION Network 26: PLC -> Scada: Vestuario: Estado (0-Desocupado / 1-Ocupado / 2-Falla reconocida / 3-Falla nueva)
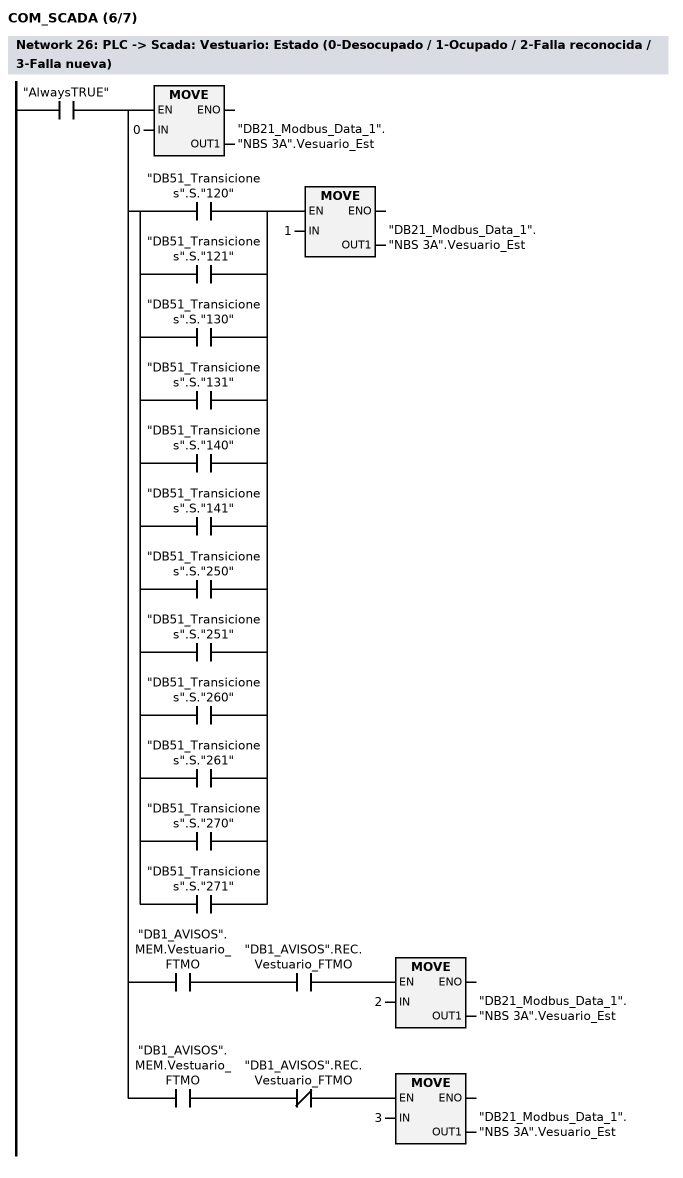
   RUNG wire#powerrail
      Contact( "AlwaysTRUE" )
      wire#w1
      Move(in := 0, out1 => "DB21_Modbus_Data_1"."NBS 3A".Vesuario_Est)
   END_RUNG
   RUNG wire#w1
      Contact( "DB51_Transiciones".S."120" )
      wire#w2
      Move(in := 1, out1 => "DB21_Modbus_Data_1"."NBS 3A".Vesuario_Est)
   END_RUNG
   RUNG wire#w1
      Contact( "DB51_Transiciones".S."121" )
   END_RUNG wire#w2
   RUNG wire#w1
      Contact( "DB51_Transiciones".S."130" )
   END_RUNG wire#w2
   RUNG wire#w1
      Contact( "DB51_Transiciones".S."131" )
   END_RUNG wire#w2
   RUNG wire#w1
      Contact( "DB51_Transiciones".S."140" )
   END_RUNG wire#w2
   RUNG wire#w1
      Contact( "DB51_Transiciones".S."141" )
   END_RUNG wire#w2
   RUNG wire#w1
      Contact( "DB51_Transiciones".S."250" )
   END_RUNG wire#w2
   RUNG wire#w1
      Contact( "DB51_Transiciones".S."251" )
   END_RUNG wire#w2
   RUNG wire#w1
      Contact( "DB51_Transiciones".S."260" )
   END_RUNG wire#w2
   RUNG wire#w1
      Contact( "DB51_Transiciones".S."261" )
   END_RUNG wire#w2
   RUNG wire#w1
      Contact( "DB51_Transiciones".S."270" )
   END_RUNG wire#w2
   RUNG wire#w1
      Contact( "DB51_Transiciones".S."271" )
   END_RUNG wire#w2
   RUNG wire#w1
      Contact( "DB1_AVISOS".MEM.Vestuario_FTMO )
      Contact( "DB1_AVISOS".REC.Vestuario_FTMO )
      Move(in := 2, out1 => "DB21_Modbus_Data_1"."NBS 3A".Vesuario_Est)
   END_RUNG
   RUNG wire#w1
      Contact( "DB1_AVISOS".MEM.Vestuario_FTMO )
      I_Contact( "DB1_AVISOS".REC.Vestuario_FTMO )
      Move(in := 3, out1 => "DB21_Modbus_Data_1"."NBS 3A".Vesuario_Est)
   END_RUNG
   // the same network as SCL:
   IF "AlwaysTRUE" THEN "DB21_Modbus_Data_1"."NBS 3A".Vesuario_Est := 0; END_IF;
   IF "AlwaysTRUE" AND ("DB51_Transiciones".S."120" OR "DB51_Transiciones".S."121" OR "DB51_Transiciones".S."130" OR "DB51_Transiciones".S."131" OR "DB51_Transiciones".S."140" OR "DB51_Transiciones".S."141" OR "DB51_Transiciones".S."250" OR "DB51_Transiciones".S."251" OR "DB51_Transiciones".S."260" OR "DB51_Transiciones".S."261" OR "DB51_Transiciones".S."270" OR "DB51_Transiciones".S."271") THEN
       "DB21_Modbus_Data_1"."NBS 3A".Vesuario_Est := 1;
   END_IF;
   IF "AlwaysTRUE" AND "DB1_AVISOS".MEM.Vestuario_FTMO AND "DB1_AVISOS".REC.Vestuario_FTMO THEN
       "DB21_Modbus_Data_1"."NBS 3A".Vesuario_Est := 2;
   END_IF;
   IF "AlwaysTRUE" AND "DB1_AVISOS".MEM.Vestuario_FTMO AND NOT "DB1_AVISOS".REC.Vestuario_FTMO THEN
       "DB21_Modbus_Data_1"."NBS 3A".Vesuario_Est := 3;
   END_IF;
END_REGION

REGION Network 27: PLC -> Scada: Ducha: Estado (0-Desocupada / 1-Ocupada / 2-Falla reconocida / 3-Falla nueva)
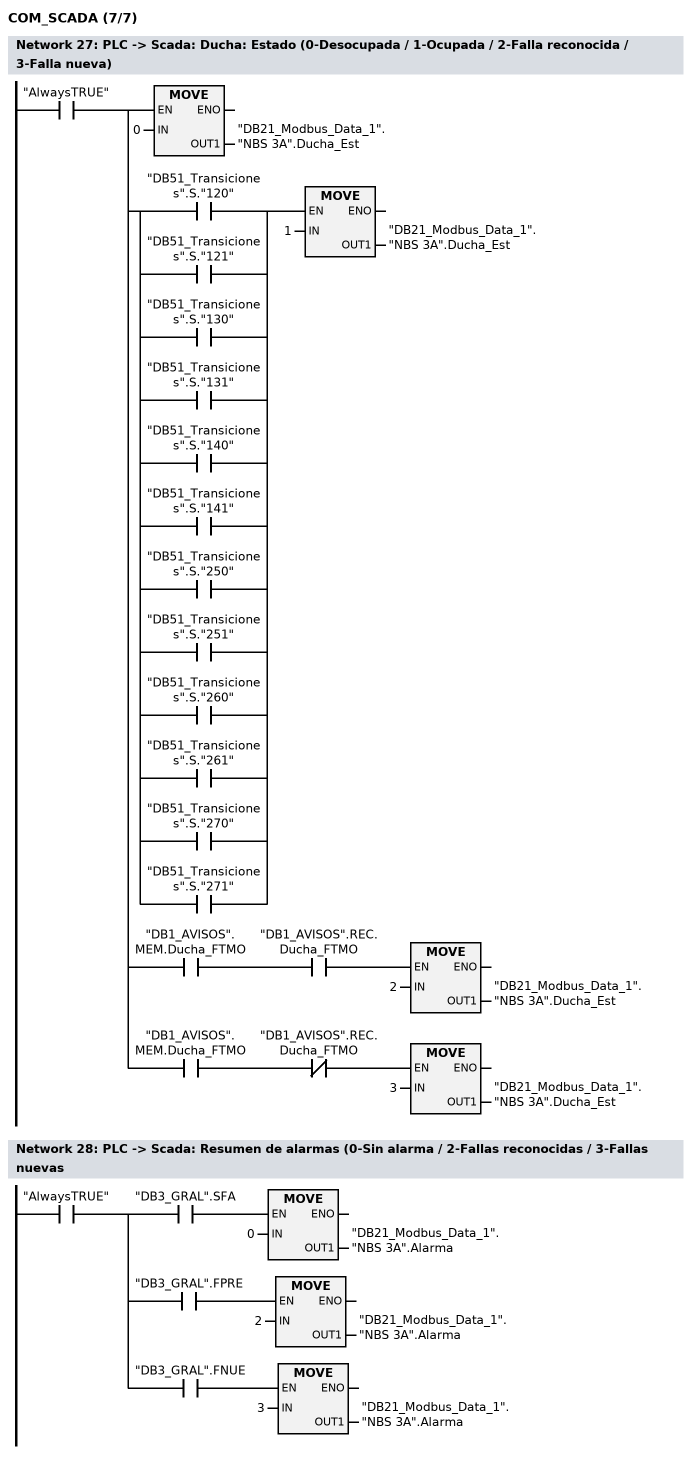
   RUNG wire#powerrail
      Contact( "AlwaysTRUE" )
      wire#w1
      Move(in := 0, out1 => "DB21_Modbus_Data_1"."NBS 3A".Ducha_Est)
   END_RUNG
   RUNG wire#w1
      Contact( "DB51_Transiciones".S."120" )
      wire#w2
      Move(in := 1, out1 => "DB21_Modbus_Data_1"."NBS 3A".Ducha_Est)
   END_RUNG
   RUNG wire#w1
      Contact( "DB51_Transiciones".S."121" )
   END_RUNG wire#w2
   RUNG wire#w1
      Contact( "DB51_Transiciones".S."130" )
   END_RUNG wire#w2
   RUNG wire#w1
      Contact( "DB51_Transiciones".S."131" )
   END_RUNG wire#w2
   RUNG wire#w1
      Contact( "DB51_Transiciones".S."140" )
   END_RUNG wire#w2
   RUNG wire#w1
      Contact( "DB51_Transiciones".S."141" )
   END_RUNG wire#w2
   RUNG wire#w1
      Contact( "DB51_Transiciones".S."250" )
   END_RUNG wire#w2
   RUNG wire#w1
      Contact( "DB51_Transiciones".S."251" )
   END_RUNG wire#w2
   RUNG wire#w1
      Contact( "DB51_Transiciones".S."260" )
   END_RUNG wire#w2
   RUNG wire#w1
      Contact( "DB51_Transiciones".S."261" )
   END_RUNG wire#w2
   RUNG wire#w1
      Contact( "DB51_Transiciones".S."270" )
   END_RUNG wire#w2
   RUNG wire#w1
      Contact( "DB51_Transiciones".S."271" )
   END_RUNG wire#w2
   RUNG wire#w1
      Contact( "DB1_AVISOS".MEM.Ducha_FTMO )
      Contact( "DB1_AVISOS".REC.Ducha_FTMO )
      Move(in := 2, out1 => "DB21_Modbus_Data_1"."NBS 3A".Ducha_Est)
   END_RUNG
   RUNG wire#w1
      Contact( "DB1_AVISOS".MEM.Ducha_FTMO )
      I_Contact( "DB1_AVISOS".REC.Ducha_FTMO )
      Move(in := 3, out1 => "DB21_Modbus_Data_1"."NBS 3A".Ducha_Est)
   END_RUNG
   // the same network as SCL:
   IF "AlwaysTRUE" THEN "DB21_Modbus_Data_1"."NBS 3A".Ducha_Est := 0; END_IF;
   IF "AlwaysTRUE" AND ("DB51_Transiciones".S."120" OR "DB51_Transiciones".S."121" OR "DB51_Transiciones".S."130" OR "DB51_Transiciones".S."131" OR "DB51_Transiciones".S."140" OR "DB51_Transiciones".S."141" OR "DB51_Transiciones".S."250" OR "DB51_Transiciones".S."251" OR "DB51_Transiciones".S."260" OR "DB51_Transiciones".S."261" OR "DB51_Transiciones".S."270" OR "DB51_Transiciones".S."271") THEN
       "DB21_Modbus_Data_1"."NBS 3A".Ducha_Est := 1;
   END_IF;
   IF "AlwaysTRUE" AND "DB1_AVISOS".MEM.Ducha_FTMO AND "DB1_AVISOS".REC.Ducha_FTMO THEN
       "DB21_Modbus_Data_1"."NBS 3A".Ducha_Est := 2;
   END_IF;
   IF "AlwaysTRUE" AND "DB1_AVISOS".MEM.Ducha_FTMO AND NOT "DB1_AVISOS".REC.Ducha_FTMO THEN
       "DB21_Modbus_Data_1"."NBS 3A".Ducha_Est := 3;
   END_IF;
END_REGION

REGION Network 28: PLC -> Scada: Resumen de alarmas (0-Sin alarma / 2-Fallas reconocidas / 3-Fallas nuevas
   RUNG wire#powerrail
      Contact( "AlwaysTRUE" )
      wire#w1
      Contact( "DB3_GRAL".SFA )
      Move(in := 0, out1 => "DB21_Modbus_Data_1"."NBS 3A".Alarma)
   END_RUNG
   RUNG wire#w1
      Contact( "DB3_GRAL".FPRE )
      Move(in := 2, out1 => "DB21_Modbus_Data_1"."NBS 3A".Alarma)
   END_RUNG
   RUNG wire#w1
      Contact( "DB3_GRAL".FNUE )
      Move(in := 3, out1 => "DB21_Modbus_Data_1"."NBS 3A".Alarma)
   END_RUNG
   // the same network as SCL:
   IF "AlwaysTRUE" AND "DB3_GRAL".SFA THEN "DB21_Modbus_Data_1"."NBS 3A".Alarma := 0; END_IF;
   IF "AlwaysTRUE" AND "DB3_GRAL".FPRE THEN "DB21_Modbus_Data_1"."NBS 3A".Alarma := 2; END_IF;
   IF "AlwaysTRUE" AND "DB3_GRAL".FNUE THEN "DB21_Modbus_Data_1"."NBS 3A".Alarma := 3; END_IF;
END_REGION
END_FUNCTION

FUNCTION "CONTROL" : Void   // FC2, LAD
TITLE = Control de accesos - Busqueda de código válido
{ S7_Optimized_Access := 'TRUE' }
VERSION : 0.1
   VAR_TEMP   // added for the SCL form of the ladder/FBD networks
      _w1 : Bool;
      _w2 : Bool;
      _w3 : Bool;
   END_VAR
BEGIN

REGION Network 1: Configuración de puerto
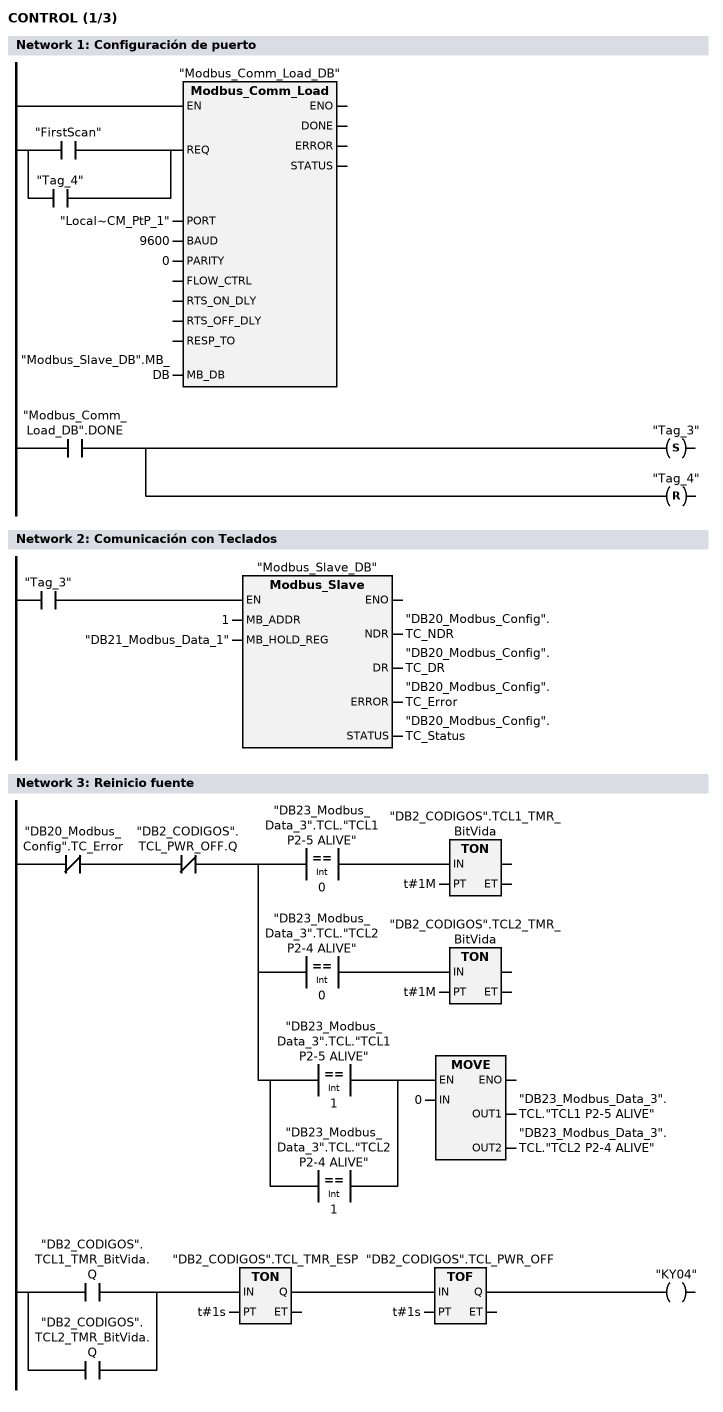
   "Modbus_Comm_Load_DB"(REQ := "FirstScan" OR "Tag_4",   // Modbus_Comm_Load
                         PORT := "Local~CM_PtP_1",
                         BAUD := 9600,
                         PARITY := 0,
                         MB_DB := "Modbus_Slave_DB".MB_DB);
   IF "Modbus_Comm_Load_DB".DONE THEN
       "Tag_3" := TRUE;
       "Tag_4" := FALSE;
   END_IF;
END_REGION

REGION Network 2: Comunicación con Teclados
   IF "Tag_3" THEN
       "Modbus_Slave_DB"(MB_ADDR := 1,   // Modbus_Slave
                         MB_HOLD_REG := "DB21_Modbus_Data_1",
                         NDR => "DB20_Modbus_Config".TC_NDR,
                         DR => "DB20_Modbus_Config".TC_DR,
                         ERROR => "DB20_Modbus_Config".TC_Error,
                         STATUS => "DB20_Modbus_Config".TC_Status);
   END_IF;
END_REGION

REGION Network 3: Reinicio fuente
   #_w1 := NOT "DB20_Modbus_Config".TC_Error AND NOT "DB2_CODIGOS".TCL_PWR_OFF.Q;
   "DB2_CODIGOS".TCL1_TMR_BitVida.TON(IN := #_w1 AND ("DB23_Modbus_Data_3".TCL."TCL1 P2-5 ALIVE" = 0),
                           PT := t#1M);
   "DB2_CODIGOS".TCL2_TMR_BitVida.TON(IN := #_w1 AND ("DB23_Modbus_Data_3".TCL."TCL2 P2-4 ALIVE" = 0),
                           PT := t#1M);
   IF #_w1 AND (("DB23_Modbus_Data_3".TCL."TCL1 P2-5 ALIVE" = 1) OR ("DB23_Modbus_Data_3".TCL."TCL2 P2-4 ALIVE" = 1)) THEN
       "DB23_Modbus_Data_3".TCL."TCL1 P2-5 ALIVE" := 0;
       "DB23_Modbus_Data_3".TCL."TCL2 P2-4 ALIVE" := 0;
   END_IF;
   "DB2_CODIGOS".TCL_TMR_ESP.TON(IN := "DB2_CODIGOS".TCL1_TMR_BitVida.Q OR "DB2_CODIGOS".TCL2_TMR_BitVida.Q,
                           PT := t#1s);
   "DB2_CODIGOS".TCL_PWR_OFF.TOF(IN := "DB2_CODIGOS".TCL_TMR_ESP.Q, PT := t#1s);
   "KY04" := "DB2_CODIGOS".TCL_PWR_OFF.Q;
END_REGION

REGION Network 4: NUevo código ingresado
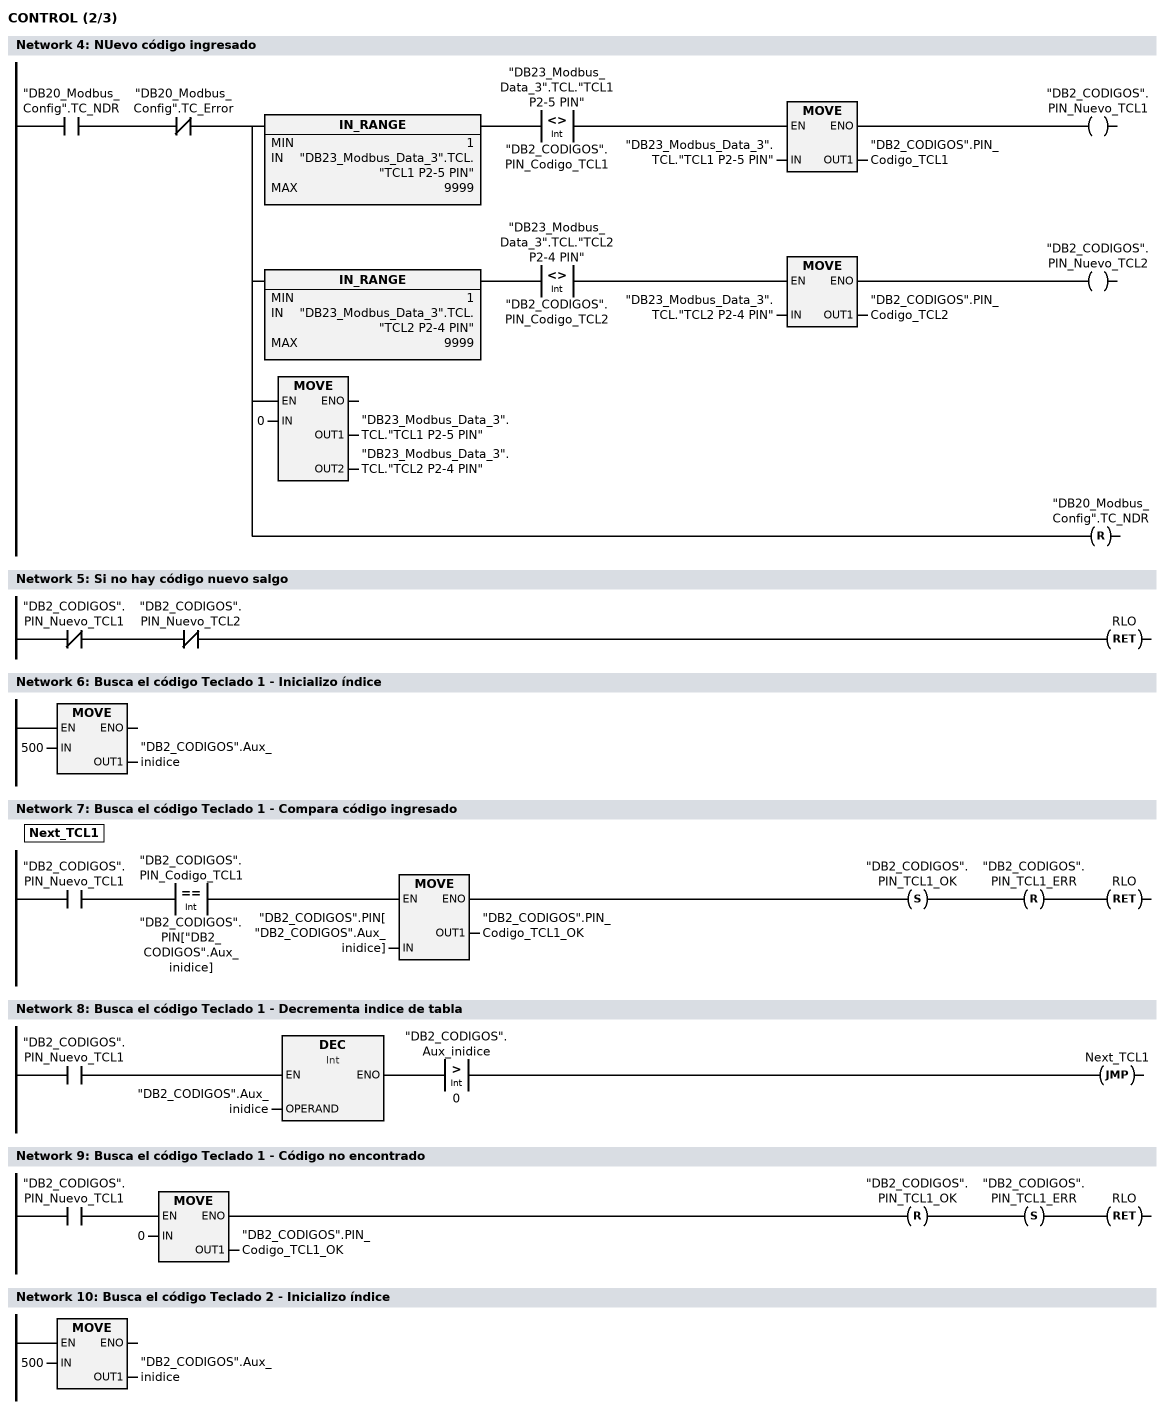
   RUNG wire#powerrail
      Contact( "DB20_Modbus_Config".TC_NDR )
      I_Contact( "DB20_Modbus_Config".TC_Error )
      wire#w1
      { S7_Templates := "SrcType := Int" } InRange(min := 1, in := "DB23_Modbus_Data_3".TCL."TCL1 P2-5 PIN", max := 9999)
      { S7_Templates := "SrcType := Int" } NE_Contact(in1 := "DB23_Modbus_Data_3".TCL."TCL1 P2-5 PIN", in2 := "DB2_CODIGOS".PIN_Codigo_TCL1)
      Move(in := "DB23_Modbus_Data_3".TCL."TCL1 P2-5 PIN", out1 => "DB2_CODIGOS".PIN_Codigo_TCL1)
      Coil( "DB2_CODIGOS".PIN_Nuevo_TCL1 )
   END_RUNG
   RUNG wire#w1
      { S7_Templates := "SrcType := Int" } InRange(min := 1, in := "DB23_Modbus_Data_3".TCL."TCL2 P2-4 PIN", max := 9999)
      { S7_Templates := "SrcType := Int" } NE_Contact(in1 := "DB23_Modbus_Data_3".TCL."TCL2 P2-4 PIN", in2 := "DB2_CODIGOS".PIN_Codigo_TCL2)
      Move(in := "DB23_Modbus_Data_3".TCL."TCL2 P2-4 PIN", out1 => "DB2_CODIGOS".PIN_Codigo_TCL2)
      Coil( "DB2_CODIGOS".PIN_Nuevo_TCL2 )
   END_RUNG
   RUNG wire#w1
      Move(in := 0, out1 => "DB23_Modbus_Data_3".TCL."TCL1 P2-5 PIN", out2 => "DB23_Modbus_Data_3".TCL."TCL2 P2-4 PIN")
   END_RUNG
   RUNG wire#w1
      R_Coil( "DB20_Modbus_Config".TC_NDR )
   END_RUNG
   // the same network as SCL:
   #_w1 := "DB20_Modbus_Config".TC_NDR AND NOT "DB20_Modbus_Config".TC_Error;
   #_w2 := #_w1 AND (1 <= "DB23_Modbus_Data_3".TCL."TCL1 P2-5 PIN") AND ("DB23_Modbus_Data_3".TCL."TCL1 P2-5 PIN" <= 9999) AND ("DB23_Modbus_Data_3".TCL."TCL1 P2-5 PIN" <> "DB2_CODIGOS".PIN_Codigo_TCL1);
   IF #_w2 THEN "DB2_CODIGOS".PIN_Codigo_TCL1 := "DB23_Modbus_Data_3".TCL."TCL1 P2-5 PIN"; END_IF;
   "DB2_CODIGOS".PIN_Nuevo_TCL1 := #_w2;
   #_w3 := #_w1 AND (1 <= "DB23_Modbus_Data_3".TCL."TCL2 P2-4 PIN") AND ("DB23_Modbus_Data_3".TCL."TCL2 P2-4 PIN" <= 9999) AND ("DB23_Modbus_Data_3".TCL."TCL2 P2-4 PIN" <> "DB2_CODIGOS".PIN_Codigo_TCL2);
   IF #_w3 THEN "DB2_CODIGOS".PIN_Codigo_TCL2 := "DB23_Modbus_Data_3".TCL."TCL2 P2-4 PIN"; END_IF;
   "DB2_CODIGOS".PIN_Nuevo_TCL2 := #_w3;
   IF #_w1 THEN
       "DB23_Modbus_Data_3".TCL."TCL1 P2-5 PIN" := 0;
       "DB23_Modbus_Data_3".TCL."TCL2 P2-4 PIN" := 0;
       "DB20_Modbus_Config".TC_NDR := FALSE;
   END_IF;
END_REGION

REGION Network 5: Si no hay código nuevo salgo
   IF NOT "DB2_CODIGOS".PIN_Nuevo_TCL1 AND NOT "DB2_CODIGOS".PIN_Nuevo_TCL2 THEN
       ENO := TRUE;
       RETURN;
   END_IF;
END_REGION

REGION Network 6: Busca el código Teclado 1 - Inicializo índice
   RUNG wire#powerrail
      Move(in := 500, out1 => "DB2_CODIGOS".Aux_inidice)
   END_RUNG
   // the same network as SCL:
   "DB2_CODIGOS".Aux_inidice := 500;
END_REGION

REGION Network 7: Busca el código Teclado 1 - Compara código ingresado
   Next_TCL1:
   #_w1 := "DB2_CODIGOS".PIN_Nuevo_TCL1 AND ("DB2_CODIGOS".PIN_Codigo_TCL1 = "DB2_CODIGOS".PIN["DB2_CODIGOS".Aux_inidice]);
   IF #_w1 THEN
       "DB2_CODIGOS".PIN_Codigo_TCL1_OK := "DB2_CODIGOS".PIN["DB2_CODIGOS".Aux_inidice];
       "DB2_CODIGOS".PIN_TCL1_OK := TRUE;
       "DB2_CODIGOS".PIN_TCL1_ERR := FALSE;
       ENO := TRUE;
       RETURN;
   END_IF;
END_REGION

REGION Network 8: Busca el código Teclado 1 - Decrementa indice de tabla
   RUNG wire#powerrail
      Contact( "DB2_CODIGOS".PIN_Nuevo_TCL1 )
      { S7_Templates := "DestType := Int" } Dec( "DB2_CODIGOS".Aux_inidice )
      { S7_Templates := "SrcType := Int" } GT_Contact(in1 := "DB2_CODIGOS".Aux_inidice, in2 := 0)
      JumpCoil( Next_TCL1 )
   END_RUNG
   // the same network as SCL:
   IF "DB2_CODIGOS".PIN_Nuevo_TCL1 THEN "DB2_CODIGOS".Aux_inidice := "DB2_CODIGOS".Aux_inidice - 1; END_IF;
   IF "DB2_CODIGOS".PIN_Nuevo_TCL1 AND ("DB2_CODIGOS".Aux_inidice > 0) THEN GOTO Next_TCL1; END_IF;
END_REGION

REGION Network 9: Busca el código Teclado 1 - Código no encontrado
   IF "DB2_CODIGOS".PIN_Nuevo_TCL1 THEN
       "DB2_CODIGOS".PIN_Codigo_TCL1_OK := 0;
       "DB2_CODIGOS".PIN_TCL1_OK := FALSE;
       "DB2_CODIGOS".PIN_TCL1_ERR := TRUE;
       ENO := TRUE;
       RETURN;
   END_IF;
END_REGION

REGION Network 10: Busca el código Teclado 2 - Inicializo índice
   RUNG wire#powerrail
      Move(in := 500, out1 => "DB2_CODIGOS".Aux_inidice)
   END_RUNG
   // the same network as SCL:
   "DB2_CODIGOS".Aux_inidice := 500;
END_REGION

REGION Network 11: Busca el código Teclado 2 - Compara código ingresado
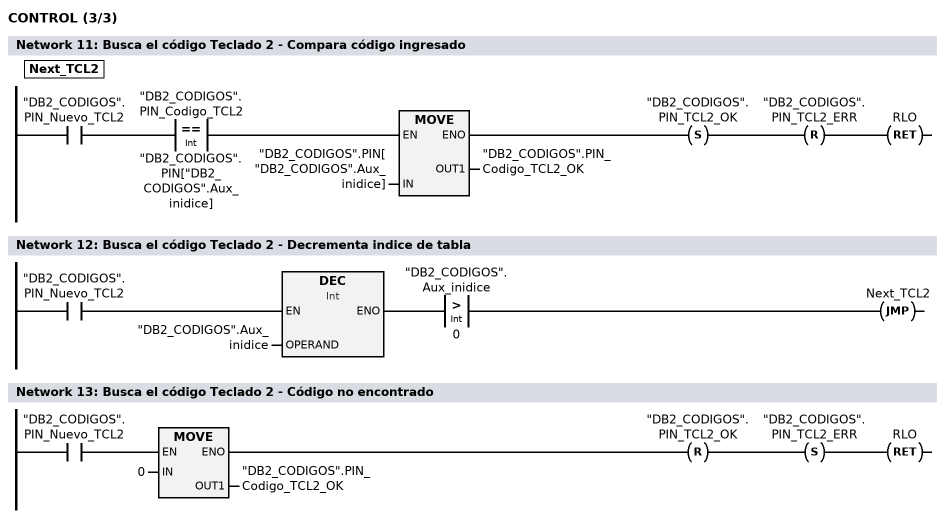
   Next_TCL2:
   #_w1 := "DB2_CODIGOS".PIN_Nuevo_TCL2 AND ("DB2_CODIGOS".PIN_Codigo_TCL2 = "DB2_CODIGOS".PIN["DB2_CODIGOS".Aux_inidice]);
   IF #_w1 THEN
       "DB2_CODIGOS".PIN_Codigo_TCL2_OK := "DB2_CODIGOS".PIN["DB2_CODIGOS".Aux_inidice];
       "DB2_CODIGOS".PIN_TCL2_OK := TRUE;
       "DB2_CODIGOS".PIN_TCL2_ERR := FALSE;
       ENO := TRUE;
       RETURN;
   END_IF;
END_REGION

REGION Network 12: Busca el código Teclado 2 - Decrementa indice de tabla
   RUNG wire#powerrail
      Contact( "DB2_CODIGOS".PIN_Nuevo_TCL2 )
      { S7_Templates := "DestType := Int" } Dec( "DB2_CODIGOS".Aux_inidice )
      { S7_Templates := "SrcType := Int" } GT_Contact(in1 := "DB2_CODIGOS".Aux_inidice, in2 := 0)
      JumpCoil( Next_TCL2 )
   END_RUNG
   // the same network as SCL:
   IF "DB2_CODIGOS".PIN_Nuevo_TCL2 THEN "DB2_CODIGOS".Aux_inidice := "DB2_CODIGOS".Aux_inidice - 1; END_IF;
   IF "DB2_CODIGOS".PIN_Nuevo_TCL2 AND ("DB2_CODIGOS".Aux_inidice > 0) THEN GOTO Next_TCL2; END_IF;
END_REGION

REGION Network 13: Busca el código Teclado 2 - Código no encontrado
   IF "DB2_CODIGOS".PIN_Nuevo_TCL2 THEN
       "DB2_CODIGOS".PIN_Codigo_TCL2_OK := 0;
       "DB2_CODIGOS".PIN_TCL2_OK := FALSE;
       "DB2_CODIGOS".PIN_TCL2_ERR := TRUE;
       ENO := TRUE;
       RETURN;
   END_IF;
END_REGION
END_FUNCTION

FUNCTION "TRAN" : Void   // FC3, LAD
TITLE = Transiciones
{ S7_Optimized_Access := 'TRUE' }
AUTHOR : IGLP
VERSION : 0.1
BEGIN

REGION Network 1: Tiempo excedido puerta abierta
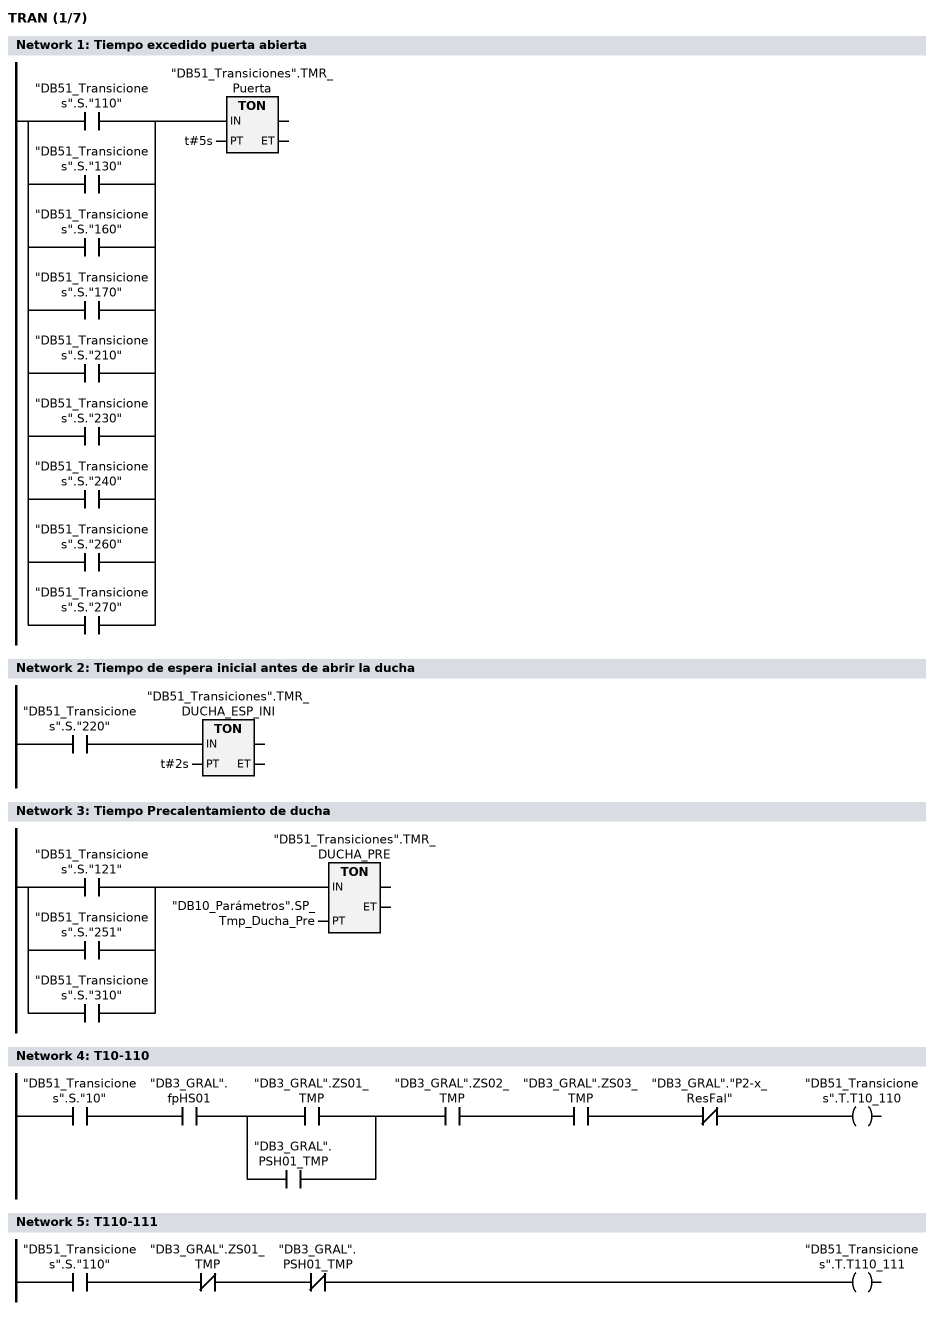
   "DB51_Transiciones".TMR_Puerta.TON(IN := "DB51_Transiciones".S."110" OR "DB51_Transiciones".S."130" OR "DB51_Transiciones".S."160" OR "DB51_Transiciones".S."170" OR "DB51_Transiciones".S."210" OR "DB51_Transiciones".S."230" OR "DB51_Transiciones".S."240" OR "DB51_Transiciones".S."260" OR "DB51_Transiciones".S."270",
                           PT := t#5s);
END_REGION

REGION Network 2: Tiempo de espera inicial antes de abrir la ducha
   "DB51_Transiciones".TMR_DUCHA_ESP_INI.TON(IN := "DB51_Transiciones".S."220", PT := t#2s);
END_REGION

REGION Network 3: Tiempo Precalentamiento de ducha
   "DB51_Transiciones".TMR_DUCHA_PRE.TON(IN := "DB51_Transiciones".S."121" OR "DB51_Transiciones".S."251" OR "DB51_Transiciones".S."310",
                           PT := "DB10_Parámetros".SP_Tmp_Ducha_Pre);
END_REGION

REGION Network 4: T10-110
   RUNG wire#powerrail
      Contact( "DB51_Transiciones".S."10" )
      Contact( "DB3_GRAL".fpHS01 )
      wire#w1
      Contact( "DB3_GRAL".ZS01_TMP )
      wire#w2
      Contact( "DB3_GRAL".ZS02_TMP )
      Contact( "DB3_GRAL".ZS03_TMP )
      I_Contact( "DB3_GRAL"."P2-x_ResFal" )
      Coil( "DB51_Transiciones".T.T10_110 )
   END_RUNG
   RUNG wire#w1
      Contact( "DB3_GRAL".PSH01_TMP )
   END_RUNG wire#w2
   // the same network as SCL:
   "DB51_Transiciones".T.T10_110 := "DB51_Transiciones".S."10" AND "DB3_GRAL".fpHS01 AND ("DB3_GRAL".ZS01_TMP OR "DB3_GRAL".PSH01_TMP) AND "DB3_GRAL".ZS02_TMP AND "DB3_GRAL".ZS03_TMP AND NOT "DB3_GRAL"."P2-x_ResFal";
END_REGION

REGION Network 5: T110-111
   RUNG wire#powerrail
      Contact( "DB51_Transiciones".S."110" )
      I_Contact( "DB3_GRAL".ZS01_TMP )
      I_Contact( "DB3_GRAL".PSH01_TMP )
      Coil( "DB51_Transiciones".T.T110_111 )
   END_RUNG
   // the same network as SCL:
   "DB51_Transiciones".T.T110_111 := "DB51_Transiciones".S."110" AND NOT "DB3_GRAL".ZS01_TMP AND NOT "DB3_GRAL".PSH01_TMP;
END_REGION

REGION Network 6: T110-10
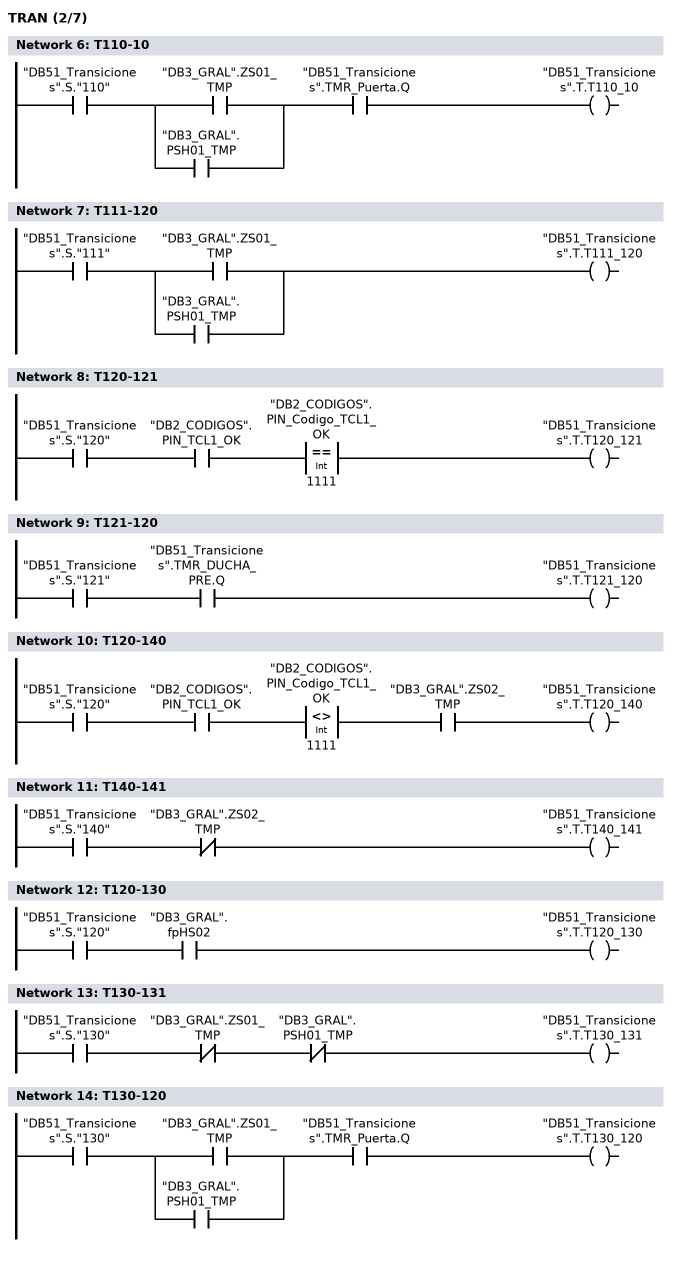
   RUNG wire#powerrail
      Contact( "DB51_Transiciones".S."110" )
      wire#w1
      Contact( "DB3_GRAL".ZS01_TMP )
      wire#w2
      Contact( "DB51_Transiciones".TMR_Puerta.Q )
      Coil( "DB51_Transiciones".T.T110_10 )
   END_RUNG
   RUNG wire#w1
      Contact( "DB3_GRAL".PSH01_TMP )
   END_RUNG wire#w2
   // the same network as SCL:
   "DB51_Transiciones".T.T110_10 := "DB51_Transiciones".S."110" AND ("DB3_GRAL".ZS01_TMP OR "DB3_GRAL".PSH01_TMP) AND "DB51_Transiciones".TMR_Puerta.Q;
END_REGION

REGION Network 7: T111-120
   RUNG wire#powerrail
      Contact( "DB51_Transiciones".S."111" )
      wire#w1
      Contact( "DB3_GRAL".ZS01_TMP )
      wire#w2
      Coil( "DB51_Transiciones".T.T111_120 )
   END_RUNG
   RUNG wire#w1
      Contact( "DB3_GRAL".PSH01_TMP )
   END_RUNG wire#w2
   // the same network as SCL:
   "DB51_Transiciones".T.T111_120 := "DB51_Transiciones".S."111" AND ("DB3_GRAL".ZS01_TMP OR "DB3_GRAL".PSH01_TMP);
END_REGION

REGION Network 8: T120-121
   RUNG wire#powerrail
      Contact( "DB51_Transiciones".S."120" )
      Contact( "DB2_CODIGOS".PIN_TCL1_OK )
      { S7_Templates := "SrcType := Int" } EQ_Contact(in1 := "DB2_CODIGOS".PIN_Codigo_TCL1_OK, in2 := 1111)
      Coil( "DB51_Transiciones".T.T120_121 )
   END_RUNG
   // the same network as SCL:
   "DB51_Transiciones".T.T120_121 := "DB51_Transiciones".S."120" AND "DB2_CODIGOS".PIN_TCL1_OK AND ("DB2_CODIGOS".PIN_Codigo_TCL1_OK = 1111);
END_REGION

REGION Network 9: T121-120
   RUNG wire#powerrail
      Contact( "DB51_Transiciones".S."121" )
      Contact( "DB51_Transiciones".TMR_DUCHA_PRE.Q )
      Coil( "DB51_Transiciones".T.T121_120 )
   END_RUNG
   // the same network as SCL:
   "DB51_Transiciones".T.T121_120 := "DB51_Transiciones".S."121" AND "DB51_Transiciones".TMR_DUCHA_PRE.Q;
END_REGION

REGION Network 10: T120-140
   RUNG wire#powerrail
      Contact( "DB51_Transiciones".S."120" )
      Contact( "DB2_CODIGOS".PIN_TCL1_OK )
      { S7_Templates := "SrcType := Int" } NE_Contact(in1 := "DB2_CODIGOS".PIN_Codigo_TCL1_OK, in2 := 1111)
      Contact( "DB3_GRAL".ZS02_TMP )
      Coil( "DB51_Transiciones".T.T120_140 )
   END_RUNG
   // the same network as SCL:
   "DB51_Transiciones".T.T120_140 := "DB51_Transiciones".S."120" AND "DB2_CODIGOS".PIN_TCL1_OK AND ("DB2_CODIGOS".PIN_Codigo_TCL1_OK <> 1111) AND "DB3_GRAL".ZS02_TMP;
END_REGION

REGION Network 11: T140-141
   RUNG wire#powerrail
      Contact( "DB51_Transiciones".S."140" )
      I_Contact( "DB3_GRAL".ZS02_TMP )
      Coil( "DB51_Transiciones".T.T140_141 )
   END_RUNG
   // the same network as SCL:
   "DB51_Transiciones".T.T140_141 := "DB51_Transiciones".S."140" AND NOT "DB3_GRAL".ZS02_TMP;
END_REGION

REGION Network 12: T120-130
   RUNG wire#powerrail
      Contact( "DB51_Transiciones".S."120" )
      Contact( "DB3_GRAL".fpHS02 )
      Coil( "DB51_Transiciones".T.T120_130 )
   END_RUNG
   // the same network as SCL:
   "DB51_Transiciones".T.T120_130 := "DB51_Transiciones".S."120" AND "DB3_GRAL".fpHS02;
END_REGION

REGION Network 13: T130-131
   RUNG wire#powerrail
      Contact( "DB51_Transiciones".S."130" )
      I_Contact( "DB3_GRAL".ZS01_TMP )
      I_Contact( "DB3_GRAL".PSH01_TMP )
      Coil( "DB51_Transiciones".T.T130_131 )
   END_RUNG
   // the same network as SCL:
   "DB51_Transiciones".T.T130_131 := "DB51_Transiciones".S."130" AND NOT "DB3_GRAL".ZS01_TMP AND NOT "DB3_GRAL".PSH01_TMP;
END_REGION

REGION Network 14: T130-120
   RUNG wire#powerrail
      Contact( "DB51_Transiciones".S."130" )
      wire#w1
      Contact( "DB3_GRAL".ZS01_TMP )
      wire#w2
      Contact( "DB51_Transiciones".TMR_Puerta.Q )
      Coil( "DB51_Transiciones".T.T130_120 )
   END_RUNG
   RUNG wire#w1
      Contact( "DB3_GRAL".PSH01_TMP )
   END_RUNG wire#w2
   // the same network as SCL:
   "DB51_Transiciones".T.T130_120 := "DB51_Transiciones".S."130" AND ("DB3_GRAL".ZS01_TMP OR "DB3_GRAL".PSH01_TMP) AND "DB51_Transiciones".TMR_Puerta.Q;
END_REGION

REGION Network 15: T131-10
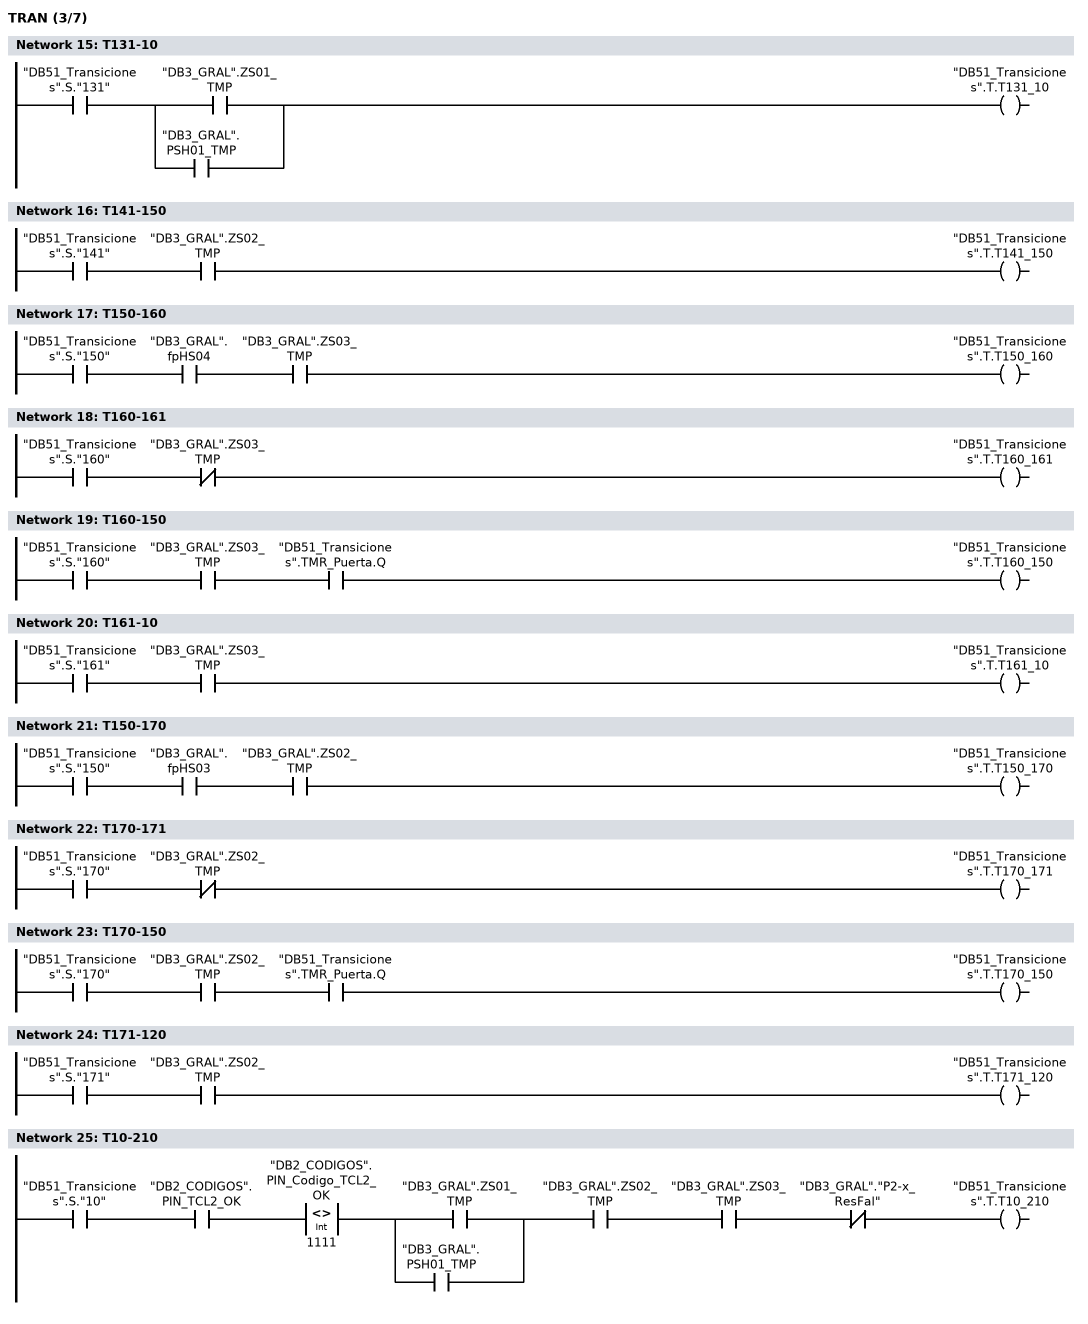
   RUNG wire#powerrail
      Contact( "DB51_Transiciones".S."131" )
      wire#w1
      Contact( "DB3_GRAL".ZS01_TMP )
      wire#w2
      Coil( "DB51_Transiciones".T.T131_10 )
   END_RUNG
   RUNG wire#w1
      Contact( "DB3_GRAL".PSH01_TMP )
   END_RUNG wire#w2
   // the same network as SCL:
   "DB51_Transiciones".T.T131_10 := "DB51_Transiciones".S."131" AND ("DB3_GRAL".ZS01_TMP OR "DB3_GRAL".PSH01_TMP);
END_REGION

REGION Network 16: T141-150
   RUNG wire#powerrail
      Contact( "DB51_Transiciones".S."141" )
      Contact( "DB3_GRAL".ZS02_TMP )
      Coil( "DB51_Transiciones".T.T141_150 )
   END_RUNG
   // the same network as SCL:
   "DB51_Transiciones".T.T141_150 := "DB51_Transiciones".S."141" AND "DB3_GRAL".ZS02_TMP;
END_REGION

REGION Network 17: T150-160
   RUNG wire#powerrail
      Contact( "DB51_Transiciones".S."150" )
      Contact( "DB3_GRAL".fpHS04 )
      Contact( "DB3_GRAL".ZS03_TMP )
      Coil( "DB51_Transiciones".T.T150_160 )
   END_RUNG
   // the same network as SCL:
   "DB51_Transiciones".T.T150_160 := "DB51_Transiciones".S."150" AND "DB3_GRAL".fpHS04 AND "DB3_GRAL".ZS03_TMP;
END_REGION

REGION Network 18: T160-161
   RUNG wire#powerrail
      Contact( "DB51_Transiciones".S."160" )
      I_Contact( "DB3_GRAL".ZS03_TMP )
      Coil( "DB51_Transiciones".T.T160_161 )
   END_RUNG
   // the same network as SCL:
   "DB51_Transiciones".T.T160_161 := "DB51_Transiciones".S."160" AND NOT "DB3_GRAL".ZS03_TMP;
END_REGION

REGION Network 19: T160-150
   RUNG wire#powerrail
      Contact( "DB51_Transiciones".S."160" )
      Contact( "DB3_GRAL".ZS03_TMP )
      Contact( "DB51_Transiciones".TMR_Puerta.Q )
      Coil( "DB51_Transiciones".T.T160_150 )
   END_RUNG
   // the same network as SCL:
   "DB51_Transiciones".T.T160_150 := "DB51_Transiciones".S."160" AND "DB3_GRAL".ZS03_TMP AND "DB51_Transiciones".TMR_Puerta.Q;
END_REGION

REGION Network 20: T161-10
   RUNG wire#powerrail
      Contact( "DB51_Transiciones".S."161" )
      Contact( "DB3_GRAL".ZS03_TMP )
      Coil( "DB51_Transiciones".T.T161_10 )
   END_RUNG
   // the same network as SCL:
   "DB51_Transiciones".T.T161_10 := "DB51_Transiciones".S."161" AND "DB3_GRAL".ZS03_TMP;
END_REGION

REGION Network 21: T150-170
   RUNG wire#powerrail
      Contact( "DB51_Transiciones".S."150" )
      Contact( "DB3_GRAL".fpHS03 )
      Contact( "DB3_GRAL".ZS02_TMP )
      Coil( "DB51_Transiciones".T.T150_170 )
   END_RUNG
   // the same network as SCL:
   "DB51_Transiciones".T.T150_170 := "DB51_Transiciones".S."150" AND "DB3_GRAL".fpHS03 AND "DB3_GRAL".ZS02_TMP;
END_REGION

REGION Network 22: T170-171
   RUNG wire#powerrail
      Contact( "DB51_Transiciones".S."170" )
      I_Contact( "DB3_GRAL".ZS02_TMP )
      Coil( "DB51_Transiciones".T.T170_171 )
   END_RUNG
   // the same network as SCL:
   "DB51_Transiciones".T.T170_171 := "DB51_Transiciones".S."170" AND NOT "DB3_GRAL".ZS02_TMP;
END_REGION

REGION Network 23: T170-150
   RUNG wire#powerrail
      Contact( "DB51_Transiciones".S."170" )
      Contact( "DB3_GRAL".ZS02_TMP )
      Contact( "DB51_Transiciones".TMR_Puerta.Q )
      Coil( "DB51_Transiciones".T.T170_150 )
   END_RUNG
   // the same network as SCL:
   "DB51_Transiciones".T.T170_150 := "DB51_Transiciones".S."170" AND "DB3_GRAL".ZS02_TMP AND "DB51_Transiciones".TMR_Puerta.Q;
END_REGION

REGION Network 24: T171-120
   RUNG wire#powerrail
      Contact( "DB51_Transiciones".S."171" )
      Contact( "DB3_GRAL".ZS02_TMP )
      Coil( "DB51_Transiciones".T.T171_120 )
   END_RUNG
   // the same network as SCL:
   "DB51_Transiciones".T.T171_120 := "DB51_Transiciones".S."171" AND "DB3_GRAL".ZS02_TMP;
END_REGION

REGION Network 25: T10-210
   RUNG wire#powerrail
      Contact( "DB51_Transiciones".S."10" )
      Contact( "DB2_CODIGOS".PIN_TCL2_OK )
      { S7_Templates := "SrcType := Int" } NE_Contact(in1 := "DB2_CODIGOS".PIN_Codigo_TCL2_OK, in2 := 1111)
      wire#w1
      Contact( "DB3_GRAL".ZS01_TMP )
      wire#w2
      Contact( "DB3_GRAL".ZS02_TMP )
      Contact( "DB3_GRAL".ZS03_TMP )
      I_Contact( "DB3_GRAL"."P2-x_ResFal" )
      Coil( "DB51_Transiciones".T.T10_210 )
   END_RUNG
   RUNG wire#w1
      Contact( "DB3_GRAL".PSH01_TMP )
   END_RUNG wire#w2
   // the same network as SCL:
   "DB51_Transiciones".T.T10_210 := "DB51_Transiciones".S."10" AND "DB2_CODIGOS".PIN_TCL2_OK AND ("DB2_CODIGOS".PIN_Codigo_TCL2_OK <> 1111) AND ("DB3_GRAL".ZS01_TMP OR "DB3_GRAL".PSH01_TMP) AND "DB3_GRAL".ZS02_TMP AND "DB3_GRAL".ZS03_TMP AND NOT "DB3_GRAL"."P2-x_ResFal";
END_REGION

REGION Network 26: T210-211
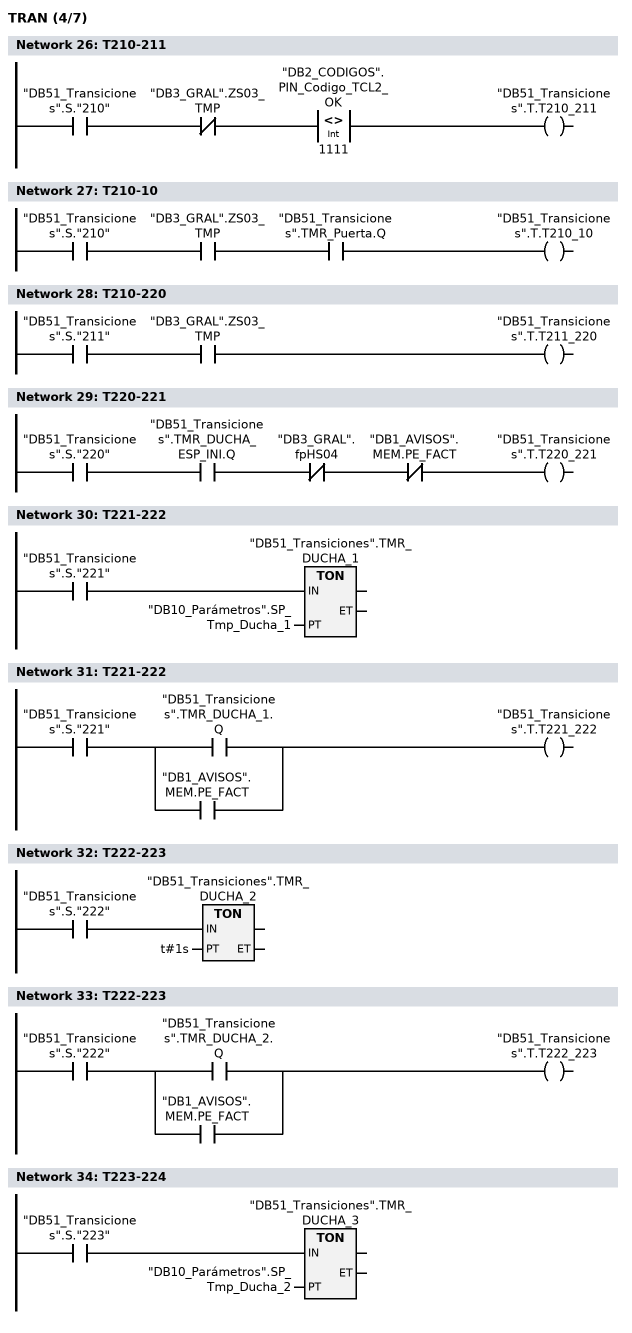
   RUNG wire#powerrail
      Contact( "DB51_Transiciones".S."210" )
      I_Contact( "DB3_GRAL".ZS03_TMP )
      { S7_Templates := "SrcType := Int" } NE_Contact(in1 := "DB2_CODIGOS".PIN_Codigo_TCL2_OK, in2 := 1111)
      Coil( "DB51_Transiciones".T.T210_211 )
   END_RUNG
   // the same network as SCL:
   "DB51_Transiciones".T.T210_211 := "DB51_Transiciones".S."210" AND NOT "DB3_GRAL".ZS03_TMP AND ("DB2_CODIGOS".PIN_Codigo_TCL2_OK <> 1111);
END_REGION

REGION Network 27: T210-10
   RUNG wire#powerrail
      Contact( "DB51_Transiciones".S."210" )
      Contact( "DB3_GRAL".ZS03_TMP )
      Contact( "DB51_Transiciones".TMR_Puerta.Q )
      Coil( "DB51_Transiciones".T.T210_10 )
   END_RUNG
   // the same network as SCL:
   "DB51_Transiciones".T.T210_10 := "DB51_Transiciones".S."210" AND "DB3_GRAL".ZS03_TMP AND "DB51_Transiciones".TMR_Puerta.Q;
END_REGION

REGION Network 28: T210-220
   RUNG wire#powerrail
      Contact( "DB51_Transiciones".S."211" )
      Contact( "DB3_GRAL".ZS03_TMP )
      Coil( "DB51_Transiciones".T.T211_220 )
   END_RUNG
   // the same network as SCL:
   "DB51_Transiciones".T.T211_220 := "DB51_Transiciones".S."211" AND "DB3_GRAL".ZS03_TMP;
END_REGION

REGION Network 29: T220-221
   RUNG wire#powerrail
      Contact( "DB51_Transiciones".S."220" )
      Contact( "DB51_Transiciones".TMR_DUCHA_ESP_INI.Q )
      I_Contact( "DB3_GRAL".fpHS04 )
      I_Contact( "DB1_AVISOS".MEM.PE_FACT )
      Coil( "DB51_Transiciones".T.T220_221 )
   END_RUNG
   // the same network as SCL:
   "DB51_Transiciones".T.T220_221 := "DB51_Transiciones".S."220" AND "DB51_Transiciones".TMR_DUCHA_ESP_INI.Q AND NOT "DB3_GRAL".fpHS04 AND NOT "DB1_AVISOS".MEM.PE_FACT;
END_REGION

REGION Network 30: T221-222
   "DB51_Transiciones".TMR_DUCHA_1.TON(IN := "DB51_Transiciones".S."221",
                           PT := "DB10_Parámetros".SP_Tmp_Ducha_1);
END_REGION

REGION Network 31: T221-222
   RUNG wire#powerrail
      Contact( "DB51_Transiciones".S."221" )
      wire#w1
      Contact( "DB51_Transiciones".TMR_DUCHA_1.Q )
      wire#w2
      Coil( "DB51_Transiciones".T.T221_222 )
   END_RUNG
   RUNG wire#w1
      Contact( "DB1_AVISOS".MEM.PE_FACT )
   END_RUNG wire#w2
   // the same network as SCL:
   "DB51_Transiciones".T.T221_222 := "DB51_Transiciones".S."221" AND ("DB51_Transiciones".TMR_DUCHA_1.Q OR "DB1_AVISOS".MEM.PE_FACT);
END_REGION

REGION Network 32: T222-223
   "DB51_Transiciones".TMR_DUCHA_2.TON(IN := "DB51_Transiciones".S."222", PT := t#1s);
END_REGION

REGION Network 33: T222-223
   RUNG wire#powerrail
      Contact( "DB51_Transiciones".S."222" )
      wire#w1
      Contact( "DB51_Transiciones".TMR_DUCHA_2.Q )
      wire#w2
      Coil( "DB51_Transiciones".T.T222_223 )
   END_RUNG
   RUNG wire#w1
      Contact( "DB1_AVISOS".MEM.PE_FACT )
   END_RUNG wire#w2
   // the same network as SCL:
   "DB51_Transiciones".T.T222_223 := "DB51_Transiciones".S."222" AND ("DB51_Transiciones".TMR_DUCHA_2.Q OR "DB1_AVISOS".MEM.PE_FACT);
END_REGION

REGION Network 34: T223-224
   "DB51_Transiciones".TMR_DUCHA_3.TON(IN := "DB51_Transiciones".S."223",
                           PT := "DB10_Parámetros".SP_Tmp_Ducha_2);
END_REGION

REGION Network 35: T223-224
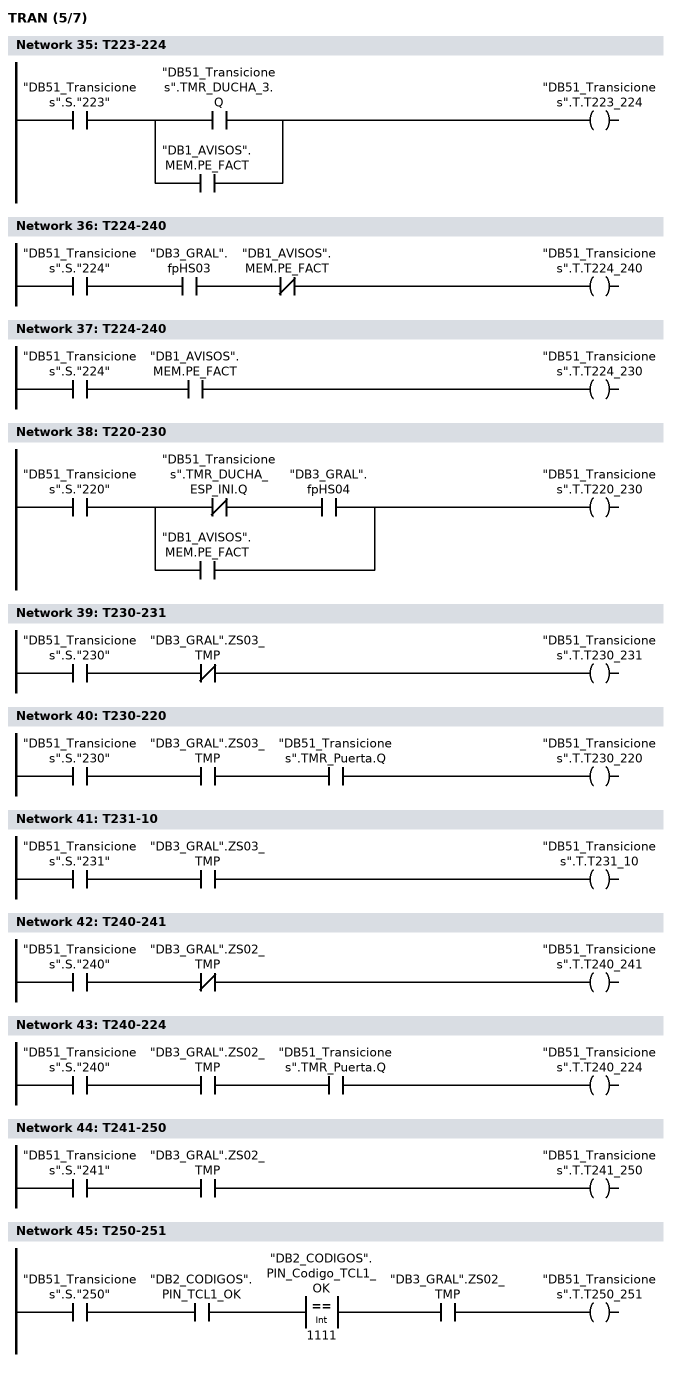
   RUNG wire#powerrail
      Contact( "DB51_Transiciones".S."223" )
      wire#w1
      Contact( "DB51_Transiciones".TMR_DUCHA_3.Q )
      wire#w2
      Coil( "DB51_Transiciones".T.T223_224 )
   END_RUNG
   RUNG wire#w1
      Contact( "DB1_AVISOS".MEM.PE_FACT )
   END_RUNG wire#w2
   // the same network as SCL:
   "DB51_Transiciones".T.T223_224 := "DB51_Transiciones".S."223" AND ("DB51_Transiciones".TMR_DUCHA_3.Q OR "DB1_AVISOS".MEM.PE_FACT);
END_REGION

REGION Network 36: T224-240
   RUNG wire#powerrail
      Contact( "DB51_Transiciones".S."224" )
      Contact( "DB3_GRAL".fpHS03 )
      I_Contact( "DB1_AVISOS".MEM.PE_FACT )
      Coil( "DB51_Transiciones".T.T224_240 )
   END_RUNG
   // the same network as SCL:
   "DB51_Transiciones".T.T224_240 := "DB51_Transiciones".S."224" AND "DB3_GRAL".fpHS03 AND NOT "DB1_AVISOS".MEM.PE_FACT;
END_REGION

REGION Network 37: T224-240
   RUNG wire#powerrail
      Contact( "DB51_Transiciones".S."224" )
      Contact( "DB1_AVISOS".MEM.PE_FACT )
      Coil( "DB51_Transiciones".T.T224_230 )
   END_RUNG
   // the same network as SCL:
   "DB51_Transiciones".T.T224_230 := "DB51_Transiciones".S."224" AND "DB1_AVISOS".MEM.PE_FACT;
END_REGION

REGION Network 38: T220-230
   RUNG wire#powerrail
      Contact( "DB51_Transiciones".S."220" )
      wire#w1
      I_Contact( "DB51_Transiciones".TMR_DUCHA_ESP_INI.Q )
      Contact( "DB3_GRAL".fpHS04 )
      wire#w2
      Coil( "DB51_Transiciones".T.T220_230 )
   END_RUNG
   RUNG wire#w1
      Contact( "DB1_AVISOS".MEM.PE_FACT )
   END_RUNG wire#w2
   // the same network as SCL:
   "DB51_Transiciones".T.T220_230 := "DB51_Transiciones".S."220" AND ((NOT "DB51_Transiciones".TMR_DUCHA_ESP_INI.Q AND "DB3_GRAL".fpHS04) OR "DB1_AVISOS".MEM.PE_FACT);
END_REGION

REGION Network 39: T230-231
   RUNG wire#powerrail
      Contact( "DB51_Transiciones".S."230" )
      I_Contact( "DB3_GRAL".ZS03_TMP )
      Coil( "DB51_Transiciones".T.T230_231 )
   END_RUNG
   // the same network as SCL:
   "DB51_Transiciones".T.T230_231 := "DB51_Transiciones".S."230" AND NOT "DB3_GRAL".ZS03_TMP;
END_REGION

REGION Network 40: T230-220
   RUNG wire#powerrail
      Contact( "DB51_Transiciones".S."230" )
      Contact( "DB3_GRAL".ZS03_TMP )
      Contact( "DB51_Transiciones".TMR_Puerta.Q )
      Coil( "DB51_Transiciones".T.T230_220 )
   END_RUNG
   // the same network as SCL:
   "DB51_Transiciones".T.T230_220 := "DB51_Transiciones".S."230" AND "DB3_GRAL".ZS03_TMP AND "DB51_Transiciones".TMR_Puerta.Q;
END_REGION

REGION Network 41: T231-10
   RUNG wire#powerrail
      Contact( "DB51_Transiciones".S."231" )
      Contact( "DB3_GRAL".ZS03_TMP )
      Coil( "DB51_Transiciones".T.T231_10 )
   END_RUNG
   // the same network as SCL:
   "DB51_Transiciones".T.T231_10 := "DB51_Transiciones".S."231" AND "DB3_GRAL".ZS03_TMP;
END_REGION

REGION Network 42: T240-241
   RUNG wire#powerrail
      Contact( "DB51_Transiciones".S."240" )
      I_Contact( "DB3_GRAL".ZS02_TMP )
      Coil( "DB51_Transiciones".T.T240_241 )
   END_RUNG
   // the same network as SCL:
   "DB51_Transiciones".T.T240_241 := "DB51_Transiciones".S."240" AND NOT "DB3_GRAL".ZS02_TMP;
END_REGION

REGION Network 43: T240-224
   RUNG wire#powerrail
      Contact( "DB51_Transiciones".S."240" )
      Contact( "DB3_GRAL".ZS02_TMP )
      Contact( "DB51_Transiciones".TMR_Puerta.Q )
      Coil( "DB51_Transiciones".T.T240_224 )
   END_RUNG
   // the same network as SCL:
   "DB51_Transiciones".T.T240_224 := "DB51_Transiciones".S."240" AND "DB3_GRAL".ZS02_TMP AND "DB51_Transiciones".TMR_Puerta.Q;
END_REGION

REGION Network 44: T241-250
   RUNG wire#powerrail
      Contact( "DB51_Transiciones".S."241" )
      Contact( "DB3_GRAL".ZS02_TMP )
      Coil( "DB51_Transiciones".T.T241_250 )
   END_RUNG
   // the same network as SCL:
   "DB51_Transiciones".T.T241_250 := "DB51_Transiciones".S."241" AND "DB3_GRAL".ZS02_TMP;
END_REGION

REGION Network 45: T250-251
   RUNG wire#powerrail
      Contact( "DB51_Transiciones".S."250" )
      Contact( "DB2_CODIGOS".PIN_TCL1_OK )
      { S7_Templates := "SrcType := Int" } EQ_Contact(in1 := "DB2_CODIGOS".PIN_Codigo_TCL1_OK, in2 := 1111)
      Contact( "DB3_GRAL".ZS02_TMP )
      Coil( "DB51_Transiciones".T.T250_251 )
   END_RUNG
   // the same network as SCL:
   "DB51_Transiciones".T.T250_251 := "DB51_Transiciones".S."250" AND "DB2_CODIGOS".PIN_TCL1_OK AND ("DB2_CODIGOS".PIN_Codigo_TCL1_OK = 1111) AND "DB3_GRAL".ZS02_TMP;
END_REGION

REGION Network 46: T251-250
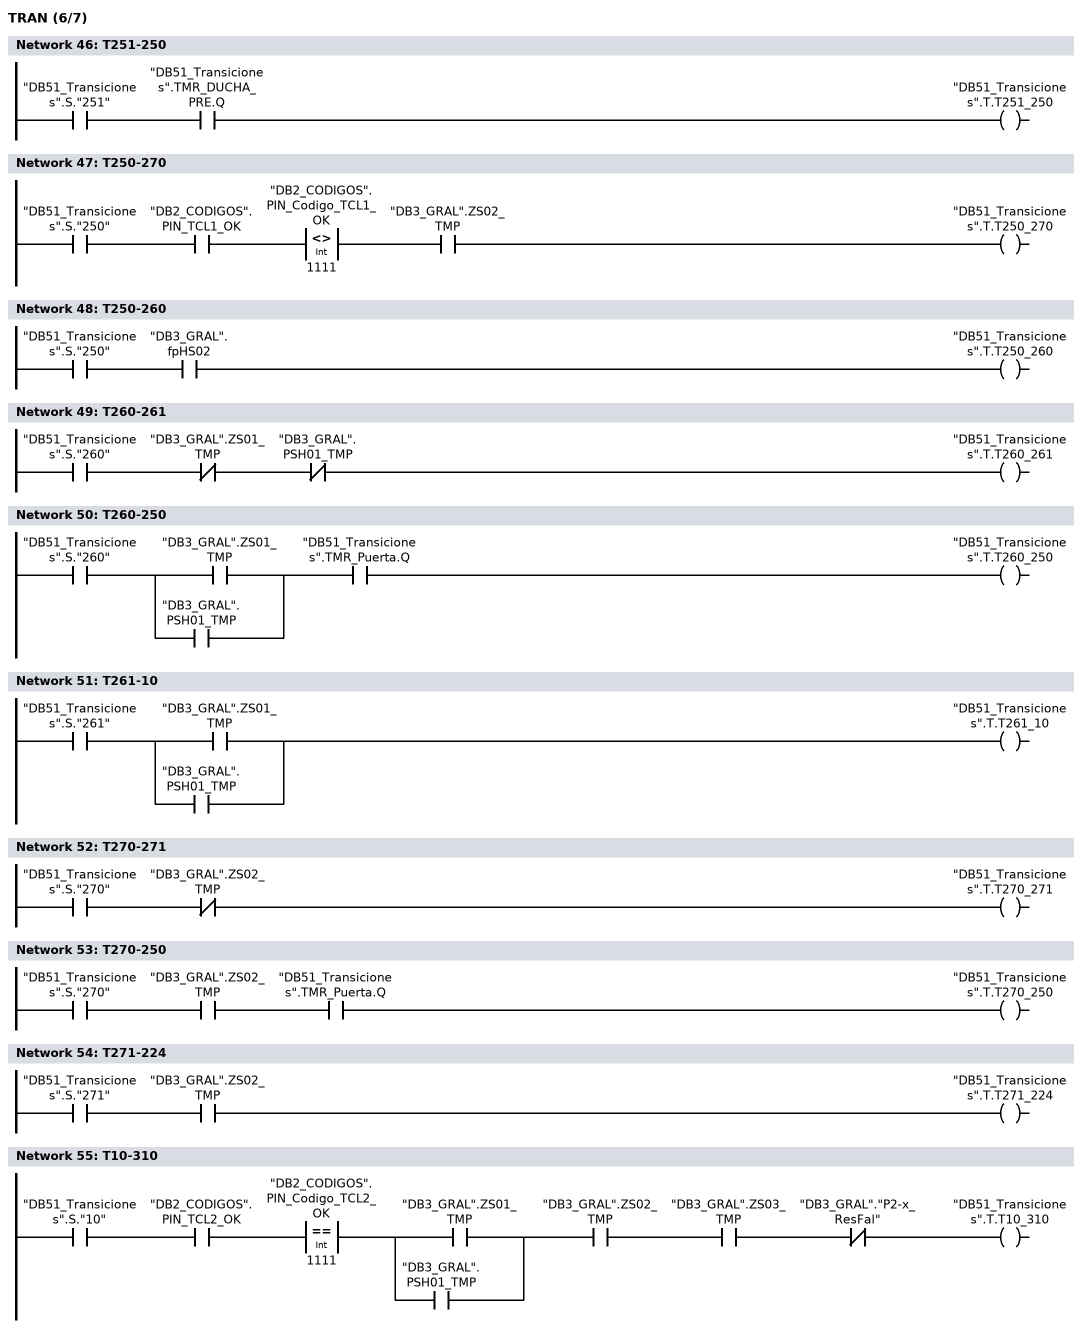
   RUNG wire#powerrail
      Contact( "DB51_Transiciones".S."251" )
      Contact( "DB51_Transiciones".TMR_DUCHA_PRE.Q )
      Coil( "DB51_Transiciones".T.T251_250 )
   END_RUNG
   // the same network as SCL:
   "DB51_Transiciones".T.T251_250 := "DB51_Transiciones".S."251" AND "DB51_Transiciones".TMR_DUCHA_PRE.Q;
END_REGION

REGION Network 47: T250-270
   RUNG wire#powerrail
      Contact( "DB51_Transiciones".S."250" )
      Contact( "DB2_CODIGOS".PIN_TCL1_OK )
      { S7_Templates := "SrcType := Int" } NE_Contact(in1 := "DB2_CODIGOS".PIN_Codigo_TCL1_OK, in2 := 1111)
      Contact( "DB3_GRAL".ZS02_TMP )
      Coil( "DB51_Transiciones".T.T250_270 )
   END_RUNG
   // the same network as SCL:
   "DB51_Transiciones".T.T250_270 := "DB51_Transiciones".S."250" AND "DB2_CODIGOS".PIN_TCL1_OK AND ("DB2_CODIGOS".PIN_Codigo_TCL1_OK <> 1111) AND "DB3_GRAL".ZS02_TMP;
END_REGION

REGION Network 48: T250-260
   RUNG wire#powerrail
      Contact( "DB51_Transiciones".S."250" )
      Contact( "DB3_GRAL".fpHS02 )
      Coil( "DB51_Transiciones".T.T250_260 )
   END_RUNG
   // the same network as SCL:
   "DB51_Transiciones".T.T250_260 := "DB51_Transiciones".S."250" AND "DB3_GRAL".fpHS02;
END_REGION

REGION Network 49: T260-261
   RUNG wire#powerrail
      Contact( "DB51_Transiciones".S."260" )
      I_Contact( "DB3_GRAL".ZS01_TMP )
      I_Contact( "DB3_GRAL".PSH01_TMP )
      Coil( "DB51_Transiciones".T.T260_261 )
   END_RUNG
   // the same network as SCL:
   "DB51_Transiciones".T.T260_261 := "DB51_Transiciones".S."260" AND NOT "DB3_GRAL".ZS01_TMP AND NOT "DB3_GRAL".PSH01_TMP;
END_REGION

REGION Network 50: T260-250
   RUNG wire#powerrail
      Contact( "DB51_Transiciones".S."260" )
      wire#w1
      Contact( "DB3_GRAL".ZS01_TMP )
      wire#w2
      Contact( "DB51_Transiciones".TMR_Puerta.Q )
      Coil( "DB51_Transiciones".T.T260_250 )
   END_RUNG
   RUNG wire#w1
      Contact( "DB3_GRAL".PSH01_TMP )
   END_RUNG wire#w2
   // the same network as SCL:
   "DB51_Transiciones".T.T260_250 := "DB51_Transiciones".S."260" AND ("DB3_GRAL".ZS01_TMP OR "DB3_GRAL".PSH01_TMP) AND "DB51_Transiciones".TMR_Puerta.Q;
END_REGION

REGION Network 51: T261-10
   RUNG wire#powerrail
      Contact( "DB51_Transiciones".S."261" )
      wire#w1
      Contact( "DB3_GRAL".ZS01_TMP )
      wire#w2
      Coil( "DB51_Transiciones".T.T261_10 )
   END_RUNG
   RUNG wire#w1
      Contact( "DB3_GRAL".PSH01_TMP )
   END_RUNG wire#w2
   // the same network as SCL:
   "DB51_Transiciones".T.T261_10 := "DB51_Transiciones".S."261" AND ("DB3_GRAL".ZS01_TMP OR "DB3_GRAL".PSH01_TMP);
END_REGION

REGION Network 52: T270-271
   RUNG wire#powerrail
      Contact( "DB51_Transiciones".S."270" )
      I_Contact( "DB3_GRAL".ZS02_TMP )
      Coil( "DB51_Transiciones".T.T270_271 )
   END_RUNG
   // the same network as SCL:
   "DB51_Transiciones".T.T270_271 := "DB51_Transiciones".S."270" AND NOT "DB3_GRAL".ZS02_TMP;
END_REGION

REGION Network 53: T270-250
   RUNG wire#powerrail
      Contact( "DB51_Transiciones".S."270" )
      Contact( "DB3_GRAL".ZS02_TMP )
      Contact( "DB51_Transiciones".TMR_Puerta.Q )
      Coil( "DB51_Transiciones".T.T270_250 )
   END_RUNG
   // the same network as SCL:
   "DB51_Transiciones".T.T270_250 := "DB51_Transiciones".S."270" AND "DB3_GRAL".ZS02_TMP AND "DB51_Transiciones".TMR_Puerta.Q;
END_REGION

REGION Network 54: T271-224
   RUNG wire#powerrail
      Contact( "DB51_Transiciones".S."271" )
      Contact( "DB3_GRAL".ZS02_TMP )
      Coil( "DB51_Transiciones".T.T271_224 )
   END_RUNG
   // the same network as SCL:
   "DB51_Transiciones".T.T271_224 := "DB51_Transiciones".S."271" AND "DB3_GRAL".ZS02_TMP;
END_REGION

REGION Network 55: T10-310
   RUNG wire#powerrail
      Contact( "DB51_Transiciones".S."10" )
      Contact( "DB2_CODIGOS".PIN_TCL2_OK )
      { S7_Templates := "SrcType := Int" } EQ_Contact(in1 := "DB2_CODIGOS".PIN_Codigo_TCL2_OK, in2 := 1111)
      wire#w1
      Contact( "DB3_GRAL".ZS01_TMP )
      wire#w2
      Contact( "DB3_GRAL".ZS02_TMP )
      Contact( "DB3_GRAL".ZS03_TMP )
      I_Contact( "DB3_GRAL"."P2-x_ResFal" )
      Coil( "DB51_Transiciones".T.T10_310 )
   END_RUNG
   RUNG wire#w1
      Contact( "DB3_GRAL".PSH01_TMP )
   END_RUNG wire#w2
   // the same network as SCL:
   "DB51_Transiciones".T.T10_310 := "DB51_Transiciones".S."10" AND "DB2_CODIGOS".PIN_TCL2_OK AND ("DB2_CODIGOS".PIN_Codigo_TCL2_OK = 1111) AND ("DB3_GRAL".ZS01_TMP OR "DB3_GRAL".PSH01_TMP) AND "DB3_GRAL".ZS02_TMP AND "DB3_GRAL".ZS03_TMP AND NOT "DB3_GRAL"."P2-x_ResFal";
END_REGION

REGION Network 56: T310-10
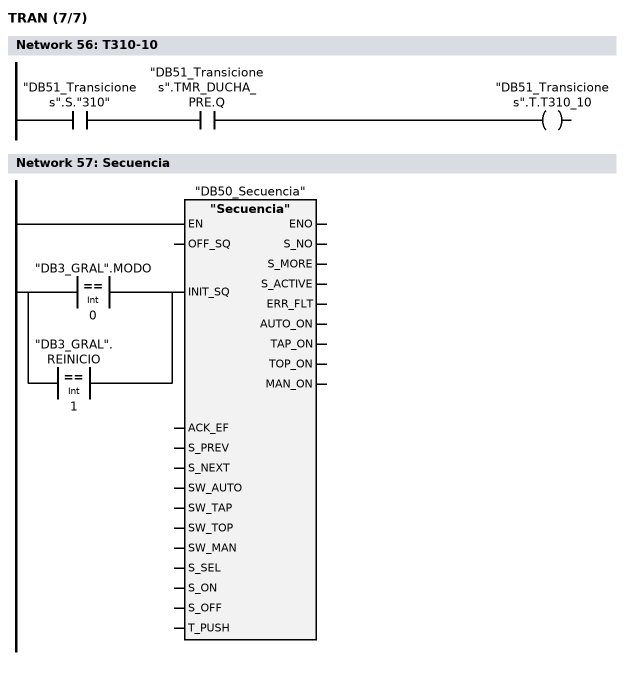
   RUNG wire#powerrail
      Contact( "DB51_Transiciones".S."310" )
      Contact( "DB51_Transiciones".TMR_DUCHA_PRE.Q )
      Coil( "DB51_Transiciones".T.T310_10 )
   END_RUNG
   // the same network as SCL:
   "DB51_Transiciones".T.T310_10 := "DB51_Transiciones".S."310" AND "DB51_Transiciones".TMR_DUCHA_PRE.Q;
END_REGION

REGION Network 57: Secuencia
   RUNG wire#powerrail
      "DB50_Secuencia"(INIT_SQ := wire#w1, OFF_SQ :=, ACK_EF :=, S_PREV :=, S_NEXT :=, SW_AUTO :=, SW_TAP :=, SW_TOP :=, SW_MAN :=, S_SEL :=, S_ON :=, S_OFF :=, T_PUSH :=, S_NO =>, S_MORE =>, S_ACTIVE =>, ERR_FLT =>, AUTO_ON =>, TAP_ON =>, TOP_ON =>, MAN_ON =>)
   END_RUNG
   RUNG wire#powerrail
      { S7_Templates := "SrcType := Int" } EQ_Contact(in1 := "DB3_GRAL".MODO, in2 := 0)
   END_RUNG wire#w1
   RUNG wire#powerrail
      { S7_Templates := "SrcType := Int" } EQ_Contact(in1 := "DB3_GRAL".REINICIO, in2 := 1)
   END_RUNG wire#w1
   // the same network as SCL:
   "DB50_Secuencia"(INIT_SQ := ("DB3_GRAL".MODO = 0) OR ("DB3_GRAL".REINICIO = 1));   // "Secuencia"
END_REGION
END_FUNCTION

FUNCTION "GRAL" : Void   // FC4, LAD
TITLE = Comandos eléctricos
{ S7_Optimized_Access := 'TRUE' }
AUTHOR : IGLP
VERSION : 0.1
   VAR_TEMP   // added for the SCL form of the ladder/FBD networks
      _w1 : Bool;
      _w2 : Bool;
   END_VAR
BEGIN

